# B&R Automation Studio project Y4_V3_1 (part 3)

#### IecCheck.st - Implementation file
```iecst
(********************************************************************
 * COPYRIGHT --
 ********************************************************************
 * Library: IecCheck
 * Author: NickE
 * Created: July 12, 2011
 ********************************************************************
 * Implementation of library IecCheck
 ********************************************************************)

(* Check divisor for DINT and UDINT division *)
FUNCTION CheckDivDWord
	IF divisor=0 THEN
		CheckDivDWord:=1;
	ELSE
		CheckDivDWord:=divisor;
	END_IF
END_FUNCTION

(* Check divisor for INT and UINT division *)
FUNCTION CheckDivWord
	IF divisor=0 THEN
		CheckDivWord:=1;
	ELSE
		CheckDivWord:=divisor;
	END_IF
END_FUNCTION

(* Check divisor for SINT and USINT division *)
FUNCTION CheckDivByte
	IF divisor=0 THEN
		CheckDivByte:=1;
	ELSE
		CheckDivByte:=divisor;
	END_IF
END_FUNCTION

(* Check divisor for REAL division *)
FUNCTION CheckDivReal
	IF divisor=0 THEN
		CheckDivReal:=1;
	ELSE
		CheckDivReal:=divisor;
	END_IF
END_FUNCTION

(* Check divisor for LREAL division *)
FUNCTION CheckDivLReal
	IF divisor=0 THEN
		CheckDivLReal:=1;
	ELSE
		CheckDivLReal:=divisor;
	END_IF
END_FUNCTION

(* Check range for array access *)
FUNCTION CheckBounds
	IF index < lower THEN
		CheckBounds := lower;
	ELSIF index > upper THEN
		CheckBounds := upper;
	ELSE
		CheckBounds := index;
	END_IF
END_FUNCTION

(* Check range for enumeration *)
FUNCTION CheckRange
	IF value < lower THEN
		CheckRange := lower;
	ELSIF value > upper THEN
		CheckRange := upper;
	ELSE
		CheckRange := value;
	END_IF
END_FUNCTION

(* Check address when reading dynamic variables *)
FUNCTION CheckReadAccess
	IF address=0 THEN
		(* TODO: Insert an appropriate code, see AutomationStudio help for further information *)
	END_IF

	CheckReadAccess:=0;
END_FUNCTION

(* Check address when writing dynamic variables *)
FUNCTION CheckWriteAccess
	IF address=0 THEN
		(* TODO: Insert an appropriate code, see AutomationStudio help for further information *)
	END_IF

	CheckWriteAccess:=0;
END_FUNCTION
```

### Library Logical/Libraries/Lib_Ashton (IEC)

#### Lib_Ashton.fun - Exported functions and function blocks
```iecst
(********************************************************************
 * COPYRIGHT --
 ********************************************************************
 * Library: Ashton
 * File: Ashton.fun
 * Author: nicke
 * Created: May 27, 2008
 ********************************************************************
 * Functions and function blocks of library Ashton
 ********************************************************************)

FUNCTION_BLOCK TrackCount (*Count Tracked pieces*)
	VAR_INPUT
		IN1 : USINT; (*Add your parameter comment*)
		IN2 : USINT; (*Add your parameter comment*)
		IN3 : USINT; (*Add your parameter comment*)
		IN4 : USINT; (*Add your parameter comment*)
		IN5 : USINT; (*Add your parameter comment*)
		IN6 : USINT; (*Add your parameter comment*)
	END_VAR
	VAR_OUTPUT
		Count : USINT; (*Add your parameter comment*)
	END_VAR
END_FUNCTION_BLOCK

FUNCTION_BLOCK Photo (*Anti bounce input filter*)
	VAR_INPUT
		SensorIN : BOOL; (*Add your parameter comment*)
		SpeedON : REAL; (*Add your parameter comment*)
		SpeedOFF : REAL; (*Add your parameter comment*)
		OverrideON : UDINT;
		OverrideOFF : UDINT;
	END_VAR
	VAR_OUTPUT
		SensorOUT : BOOL; (*Add your parameter comment*)
		PTON : TIME;
		PTOFF : TIME;
		Measured : REAL;
	END_VAR
	VAR
		Measure : CycleTime_typ;
		DelayB4ON : TON; (*Add your parameter comment*)
		DelayB4OFF : TON; (*Add your parameter comment*)
		zzEdge00000 : BOOL;
		zzEdge00001 : BOOL;
		zzEdge00002 : BOOL;
		zzEdge00003 : BOOL;
	END_VAR
END_FUNCTION_BLOCK

FUNCTION_BLOCK TrackProc (*TODO: Add your comment here*)
	VAR_INPUT
		ONStart : BOOL; (*Add your parameter comment*)
		OFFStart : BOOL; (*Add your parameter comment*)
		EStop : BOOL; (*Add your parameter comment*)
		PT_On : UDINT; (*Add your parameter comment*)
		PT_Off : UDINT; (*Add your parameter comment*)
		End : BOOL;
	END_VAR
	VAR_OUTPUT
		Out : BOOL; (*Add your parameter comment*)
	END_VAR
	VAR
		ON : TON; (*Add your parameter comment*)
		OFF : TON; (*Add your parameter comment*)
		BeforeOn : BOOL;
		BeforeOff : BOOL;
		zzEdge00000 : BOOL;
		zzEdge00001 : BOOL;
		zzEdge00002 : BOOL;
		zzEdge00003 : BOOL;
		zzEdge00004 : BOOL;
		PTOnEStop : TIME;
		PTOffEStop : TIME;
		Recover : BOOL;
		ONPT : TIME;
		OFFPT : TIME;
	END_VAR
END_FUNCTION_BLOCK

FUNCTION_BLOCK C5Restart (*Calculate Restart delay for C5R*)
	VAR_INPUT
		Start : BOOL; (*Add your parameter comment*)
		Speed : REAL; (*Add your parameter comment*)
	END_VAR
	VAR_OUTPUT
		Out : BOOL; (*Add your parameter comment*)
	END_VAR
	VAR
		TON_001 : TON; (*Add your parameter comment*)
		Preset : REAL; (*Add your parameter comment*)
	END_VAR
END_FUNCTION_BLOCK

FUNCTION_BLOCK RunTime (*Calculate system run time*)
	VAR_INPUT
		On : BOOL; (*Add your parameter comment*)
		TotReset : BOOL; (*Total Reset*)
		ShftReset : BOOL; (*Shift Reset*)
		TotMinIn : UINT; (*Total minutes In*)
		TotHrIn : UINT; (*Total hours In*)
		TotDayIn : UINT; (*Total days In*)
		TotYrIn : UINT; (*Total years In*)
		ShftMinIn : UINT; (*Shft minutes In*)
		ShftHrIn : UINT; (*Shift hours In*)
		ShftDayIn : UINT; (*Shift days In*)
		ShftYrIn : UINT; (*Shift years In*)
	END_VAR
	VAR_OUTPUT
		TotMin : UINT; (*Total Minutes*)
		TotHr : UINT; (*Total Hours*)
		TotDay : UINT; (*Total Days*)
		TotYr : UINT; (*Total Years*)
		ShftMin : UINT; (*Shift Minutes*)
		ShftHr : UINT; (*Shift Hours*)
		ShftDay : UINT; (*Shift Days*)
		ShftYr : UINT; (*Shift Years*)
	END_VAR
	VAR
		Minute : TON; (*Minute timer*)
	END_VAR
END_FUNCTION_BLOCK

FUNCTION_BLOCK GrindTime (*Calculate grind time and length*)
	VAR_INPUT
		On : BOOL; (*Start trigger*)
		TotReset : BOOL; (*Total Reset*)
		ShftReset : BOOL; (*Shift Reset*)
		Speed : REAL; (*Seaming speed*)
		Measured : REAL; (*Measured length/width*)
		TotMSIn : UINT; (*Total Milliseconds*)
		TotSecIn : UINT; (*Total Seconds*)
		TotMinIn : UINT; (*Total Minutes*)
		TotHrIn : UINT; (*Total Hours*)
		TotDayIn : UINT; (*Total Days*)
		ShftMSIn : UINT; (*Shift Milliseconds*)
		ShftSecIn : UINT; (*Shift Seconds*)
		ShftMinIn : UINT; (*Shift Minutes*)
		ShftHrIn : UINT; (*Shift Hours*)
		ShftDayIn : UINT; (*Shift Days*)
		TotMtrs1In : UDINT; (*Total Meters 1*)
		TotMtrs2In : UDINT; (*Total Meters 2*)
		TotFt1In : UDINT; (*Total Feet 1*)
		TotFt2In : UDINT; (*Total Feet 2*)
		ShftMtrs1In : UDINT; (*Shift Meters 1*)
		ShftMtrs2In : UDINT; (*Shift Meters 2*)
		ShftFt1In : UDINT; (*Shift Feet 1*)
		ShftFt2In : UDINT; (*Shift Feet 2*)
	END_VAR
	VAR_OUTPUT
		TotMS : UINT; (*Total Milliseconds*)
		TotSec : UINT; (*Total Seconds*)
		TotMin : UINT; (*Total Minutes*)
		TotHr : UINT; (*Total Hours*)
		TotDay : UINT; (*Total Days*)
		ShftMS : UINT; (*Shift Milliseconds*)
		ShftSec : UINT; (*Shift Seconds*)
		ShftMin : UINT; (*Shift Minutes*)
		ShftHr : UINT; (*Shift Hours*)
		ShftDay : UINT; (*Shift Days*)
		TotMtrs1 : UDINT; (*Total Meters 1*)
		TotMtrs2 : UDINT; (*Total Meters 2*)
		TotFt1 : UDINT; (*Total Feet 1*)
		TotFt2 : UDINT; (*Total Feet 2*)
		ShftMtrs1 : UDINT; (*Shift Meters 1*)
		ShftMtrs2 : UDINT; (*Shift Meters 2*)
		ShftFt1 : UDINT; (*Shift Feet 1*)
		ShftFt2 : UDINT; (*Shift Feet 2*)
	END_VAR
	VAR
		CurrentMS : REAL; (*Current measured length in millisec*)
		WholeSec : UINT; (*Calculated whole seconds*)
		CurrentMSUINT : UINT; (*CurrentMS in UINT*)
		WholeMSec : UINT;
		Calc3 : UINT;
		MeasuredFtUD : UDINT; (*Measured feet UDINT*)
		MeasuredUD : UDINT; (*Measured Mtrs UDINT*)
		MeasuredM : REAL; (*Measured Mtrs*)
		MeasuredFt : REAL; (*Measured feet*)
		zzEdge00000 : BOOL;
	END_VAR
END_FUNCTION_BLOCK

FUNCTION_BLOCK Center2 (*TODO: Add your comment here*)
	VAR_INPUT
		WidthIn : REAL; (*Add your parameter comment*)
		Speed : REAL; (*Add your parameter comment*)
		Centre : REAL; (*Add your parameter comment*)
	END_VAR
	VAR_OUTPUT
		PT : UDINT; (*Add your parameter comment*)
	END_VAR
	VAR
		Calc1 : REAL; (*Add your parameter comment*)
		DecTime : REAL; (*Add your parameter comment*)
		DecDist : REAL; (*Add your parameter comment*)
		PTReal : REAL; (*Add your parameter comment*)
	END_VAR
END_FUNCTION_BLOCK

FUNCTION_BLOCK Center (*TODO: Add your comment here*)
	VAR_INPUT
		WidthIn : REAL; (*Add your parameter comment*)
		Speed : REAL; (*Add your parameter comment*)
		Centre : REAL; (*Add your parameter comment*)
	END_VAR
	VAR_OUTPUT
		PT : UDINT; (*Add your parameter comment*)
	END_VAR
	VAR
		Calc1 : REAL; (*Add your parameter comment*)
		AccTime : REAL; (*Add your parameter comment*)
		AccDecDist : REAL; (*Add your parameter comment*)
		PTReal : REAL; (*Add your parameter comment*)
	END_VAR
END_FUNCTION_BLOCK

FUNCTION_BLOCK TrackBit (*Tracking Bit Controls*) (*$GROUP=User,$CAT=User,$GROUPICON=User.png,$CATICON=User.png*)
	VAR_INPUT
		FixedIN : TrackBit_Fixed_typ;
		RunBlock : BOOL;
		SolBlock : BOOL;
		Analog : FB_ANALOG_enum;
		Speed : REAL;
		SpeedAnalog : REAL;
		SpeedMatchEN : BOOL;
		SpeedMatch : REAL;
		TimeoutBlock : BOOL;
		TimeoutEN : BOOL;
		TrackDelayEN : BOOL;
		DelayPT : UDINT;
		TimeoutACK : BOOL;
		DoneIN : BOOL;
	END_VAR
	VAR_OUTPUT
		Active : BOOL;
		Done : BOOL;
		Disp : Display_enum;
		ESDisp : {REDUND_UNREPLICABLE} Display_enum;
		RunOUT : BOOL;
		SolOUT : BOOL;
		SpeedOUT : REAL;
		TimeoutOUT : BOOL;
	END_VAR
	VAR
		DelayTON : TON;
		TimeoutACKLatch : BOOL;
	END_VAR
END_FUNCTION_BLOCK

FUNCTION_BLOCK TrackingSection (*TRACKING SECTION CONTROLS*) (*$GROUP=User,$CAT=User,$GROUPICON=User.png,$CATICON=User.png*)
	VAR_INPUT
		ControlIN : BOOL;
		ESClear : BOOL;
		Cleared : BOOL;
		EMOStart : BOOL;
		Blocks : ARRAY[0..12] OF BOOL;
		BlockInhib : BOOL;
		ResES : BOOL;
		ResMan : BOOL;
		ESDispInhib : BOOL;
		IndexIN : USINT;
		WidthIN : REAL;
		LengthIN : REAL;
		BatchClearIN : BOOL;
		LongestIN : REAL;
		RowBlockIN : BOOL;
		ChangeIN : BOOL;
		ArrissUpperIN : BOOL;
		ArrissLowerIN : BOOL;
		EdgeDeleteIN : BOOL;
		VerticalBeltIN : BOOL;
	END_VAR
	VAR_OUTPUT
		FixedOUT : TrackBit_Fixed_typ;
		Blocked : BOOL;
		Busy : BOOL;
		Index : USINT;
		Width : REAL;
		Length : REAL;
		BatchClear : BOOL;
		Longest : REAL;
		RowBlock : BOOL;
		Change : BOOL;
		ArrissUpper : BOOL;
		ArrissLower : BOOL;
		EdgeDelete : BOOL;
		VerticalBelt : BOOL;
		Cycle : REAL;
		BusyDisp : Display_enum;
	END_VAR
	VAR
		CurrentTime : TIME;
		PreviousTime : TIME;
		ElapsedTime : UDINT;
		i : INT;
		zzEdge00000 : BOOL;
	END_VAR
END_FUNCTION_BLOCK

FUNCTION_BLOCK ControlFB
	VAR_INPUT
		Start : BOOL;
		Stop : BOOL;
		EStop1 : BOOL;
		EStop2 : BOOL;
		BuzzBlock : BOOL;
		StandbyBlock : BOOL;
		Auto : BOOL;
		Test : BOOL;
		ESClear : BOOL;
		Paused : BOOL;
		Alarm : BOOL;
		Warning : BOOL;
		CountIN : ARRAY[0..19] OF BOOL;
		BuzzerPT : UDINT;
		StandbyPT : UDINT;
	END_VAR
	VAR_OUTPUT
		Achieved1 : BOOL;
		Achieved2 : BOOL;
		Buzzer : BOOL;
		Empty : BOOL;
		OnLmp1 : BOOL;
		OnLmp2 : BOOL;
		GrnLmp : BOOL;
		YelLmp : BOOL;
		RedLmp : BOOL;
	END_VAR
	VAR
		BuzzerTON : TON;
		StandbyTON : TON;
		Grn : ARRAY[0..2] OF BOOL;
		Yel : ARRAY[0..2] OF BOOL;
		Red : ARRAY[0..2] OF BOOL;
		TSecOff : BOOL;
		TSecOn : BOOL;
		TSecOFF : TON;
		TSecON : TON;
		StopLatch : BOOL;
		StopDone : BOOL;
		i : USINT;
		zzEdge1 : BOOL;
		zzEdge2 : BOOL;
		zzEdge3 : BOOL;
		zzEdge4 : BOOL;
		zzEdge5 : BOOL;
		EStopStartTON : TON;
		zzEdge6 : BOOL;
		zzEdge7 : BOOL;
		zzEdge00000 : BOOL;
		zzEdge00001 : BOOL;
		zzEdge00002 : BOOL;
		zzEdge00003 : BOOL;
		zzEdge00004 : BOOL;
		zzEdge00005 : BOOL;
		zzEdge00006 : BOOL;
	END_VAR
END_FUNCTION_BLOCK

FUNCTION_BLOCK SeamersFB
	VAR_INPUT
		Enable : ARRAY[0..4] OF BOOL;
		AutoStart : ARRAY[0..4] OF BOOL;
		ESClear : BOOL;
		ControlIN : BOOL;
		EDOn : BOOL;
		TransportMode : BOOL;
		Detension : BOOL;
		Trips : ARRAY[0..24] OF BOOL;
		Float : ARRAY[0..2] OF BOOL;
		BeltsPT : UDINT;
		VacPT : UDINT;
		EDPT : UDINT;
		ExtractionPT : UDINT;
		PumpPT : ARRAY[0..4] OF UDINT;
		VacsStopPT : UDINT;
	END_VAR
	VAR_OUTPUT
		StartAllDisp : Display_enum;
		BeltOUT : ARRAY[0..12] OF BOOL;
		VacOUT : ARRAY[0..4] OF BOOL;
		EDOUT : ARRAY[0..4] OF BOOL;
		ExtractionOUT : ARRAY[0..4] OF BOOL;
		PumpOUT : ARRAY[0..2] OF BOOL;
		DoneOUT : ARRAY[0..4] OF BOOL;
	END_VAR
	VAR
		zzEdge00000 : BOOL;
		zzEdge00001 : BOOL;
		zzEdge00002 : BOOL;
		zzEdge00003 : BOOL;
		zzEdge00004 : BOOL;
		zzEdge00005 : BOOL;
		zzEdge00006 : BOOL;
		zzEdge00007 : BOOL;
		zzEdge00008 : BOOL;
		zzEdge00009 : BOOL;
		zzEdge00010 : BOOL;
		zzEdge00011 : BOOL;
		zzEdge00012 : BOOL;
		zzEdge00013 : BOOL;
		zzEdge00014 : BOOL;
		zzEdge00015 : BOOL;
		zzEdge00016 : BOOL;
		zzEdge00017 : BOOL;
		zzEdge00018 : BOOL;
		zzEdge00019 : BOOL;
		zzEdge00020 : BOOL;
		zzEdge00021 : BOOL;
		zzEdge00022 : BOOL;
		zzEdge00023 : BOOL;
		zzEdge00024 : BOOL;
		zzEdge00025 : BOOL;
		zzEdge00026 : BOOL;
		zzEdge00027 : BOOL;
		Latch : BOOL;
		LatchES : BOOL;
		Starting1 : BOOL;
		Starting2 : BOOL;
		Starting3 : BOOL;
		Starting4 : BOOL;
		Belt1TON : TON;
		Belt2TON : TON;
		Belt3TON : TON;
		Belt4TON : TON;
		Belt5TON : TON;
		Belt6TON : TON;
		Belt7TON : TON;
		Belt8TON : TON;
		Belt9TON : TON;
		Belt10TON : TON;
		Belt11TON : TON;
		Belt12TON : TON;
		ED1TON : TON;
		ED2TON : TON;
		ED3TON : TON;
		ED4TON : TON;
		Vac1TON : TON;
		Vac2TON : TON;
		Vac3TON : TON;
		Vac4TON : TON;
		Extract1TON : TON;
		Extract2TON : TON;
		Extract3TON : TON;
		Extract4TON : TON;
		Pump4TON : TON;
		Pump3TON : TON;
		Pump1TON : TON;
		Pump2TON : TON;
		i : INT;
		VacStopTON : TON;
		zzEdge00028 : BOOL;
		zzEdge00029 : BOOL;
		zzEdge00030 : BOOL;
		zzEdge00031 : BOOL;
	END_VAR
END_FUNCTION_BLOCK

FUNCTION_BLOCK InvTestFB
	VAR_INPUT
		Index : USINT;
		AutoSpeedIN : REAL;
		SpeedIN : PLInvPerm;
		TestSpeedIN : REAL;
		AnalogSpeedIN : REAL;
	END_VAR
	VAR_OUTPUT
		Run : BOOL;
		Rev : BOOL;
		Speed : REAL;
	END_VAR
END_FUNCTION_BLOCK

FUNCTION_BLOCK Batch (*ROW BUILDING CALCULATIONS*) (*$GROUP=User,$CAT=User,$GROUPICON=User.png,$CATICON=User.png*)
	VAR_INPUT
		Calculate : BOOL;
		ClearIN : BOOL;
		Building : BOOL;
		Gap : REAL;
		MaxSize : REAL;
		CenterDist : REAL;
		CenterSpeed : REAL;
		FollowingIN : ARRAY[0..9] OF REAL;
		LengthIN : REAL;
		BatchMode : BATCHING_enum;
		Type : BATCHTYPE_enum;
	END_VAR
	VAR_OUTPUT
		Longest : REAL;
		Current : REAL;
		Next : REAL;
		Done : BOOL;
		CenterPT : UDINT;
		Remaining : REAL;
	END_VAR
	VAR
		i : USINT;
		MinRemaining : REAL;
		NextSize : REAL;
		NextLengthINT : REAL;
		NextINT : REAL;
		DoubleCount : USINT;
		Center : Center;
		zzEdge00000 : BOOL;
		zzEdge00001 : BOOL;
		zzEdge00002 : BOOL;
		zzEdge00003 : BOOL;
		zzEdge00004 : BOOL;
		zzEdge00005 : BOOL;
		zzEdge00006 : BOOL;
		zzEdge00007 : BOOL;
		zzEdge00008 : BOOL;
		zzEdge00009 : BOOL;
	END_VAR
END_FUNCTION_BLOCK

FUNCTION_BLOCK SeamersSMProFB (*Seamers start up control SMPro*) (*$GROUP=User,$CAT=User,$GROUPICON=User.png,$CATICON=User.png*)
	VAR_INPUT
		Enable : ARRAY[0..4] OF BOOL;
		AutoStart : ARRAY[0..4] OF BOOL;
		ESClear : BOOL;
		ControlIN : BOOL;
		EDOn : BOOL;
		TransportMode : BOOL;
		Detension : BOOL;
		Trips : ARRAY[0..24] OF BOOL;
		Float : ARRAY[0..2] OF BOOL;
		BeltsPT : UDINT;
		VacPT : UDINT;
		EDPT : UDINT;
		ExtractionPT : UDINT;
		PumpPT : ARRAY[0..4] OF UDINT;
		VacsStopPT : UDINT;
	END_VAR
	VAR_OUTPUT
		StartAllDisp : Display_enum;
		BeltOUT : ARRAY[0..12] OF BOOL;
		VacOUT : ARRAY[0..4] OF BOOL;
		EDOUT : ARRAY[0..4] OF BOOL;
		ExtractionOUT : ARRAY[0..4] OF BOOL;
		PumpOUT : ARRAY[0..2] OF BOOL;
		DoneOUT : ARRAY[0..4] OF BOOL;
	END_VAR
	VAR
		Latch : BOOL;
		LatchES : BOOL;
		Starting1 : BOOL;
		Starting2 : BOOL;
		Belt1TON : TON;
		Belt2TON : TON;
		Belt3TON : TON;
		Belt4TON : TON;
		Belt5TON : TON;
		Belt6TON : TON;
		Belt7TON : TON;
		Belt8TON : TON;
		Belt9TON : TON;
		Belt10TON : TON;
		Belt11TON : TON;
		Belt12TON : TON;
		ED1TON : TON;
		ED2TON : TON;
		ED3TON : TON;
		ED4TON : TON;
		Vac1TON : TON;
		Vac2TON : TON;
		Vac3TON : TON;
		Vac4TON : TON;
		Extract1TON : TON;
		Extract2TON : TON;
		Extract3TON : TON;
		Extract4TON : TON;
		Pump4TON : TON;
		Pump3TON : TON;
		Pump1TON : TON;
		Pump2TON : TON;
		i : INT;
		VacStopTON : TON;
		zzEdge00000 : BOOL;
		zzEdge00001 : BOOL;
		zzEdge00002 : BOOL;
		zzEdge00003 : BOOL;
		zzEdge00004 : BOOL;
		zzEdge00005 : BOOL;
		zzEdge00006 : BOOL;
		zzEdge00007 : BOOL;
		zzEdge00008 : BOOL;
		zzEdge00009 : BOOL;
		zzEdge00010 : BOOL;
		zzEdge00011 : BOOL;
		zzEdge00012 : BOOL;
		zzEdge00013 : BOOL;
		zzEdge00014 : BOOL;
		zzEdge00015 : BOOL;
		zzEdge00016 : BOOL;
		zzEdge00017 : BOOL;
	END_VAR
END_FUNCTION_BLOCK

FUNCTION_BLOCK FlipUps (*FLIP UP ARMS CONTROL*) (*$GROUP=User,$CAT=User,$GROUPICON=User.png,$CATICON=User.png*)
	VAR_INPUT
		ActPos : REAL; (*Seamer Actual Position*)
		ArmPos : ARRAY[0..5] OF REAL; (*Arm Actual Positions*)
		Up : ARRAY[0..10] OF BOOL; (*Array for arms up reed switches*)
		i : INT; (*Index for FOR loops*)
		Down : ARRAY[0..10] OF BOOL; (*Array for arms down reed switches*)
		HiVol : BOOL; (*Mode Selection*)
		Arms : USINT; (*Number of Arms*)
		Raise : BOOL; (*Condition to raise arms*)
	END_VAR
	VAR_OUTPUT
		UpDone : BOOL; (*Selected arms up*)
		OUT : ARRAY[0..5] OF BOOL; (*Raise Arms Output*)
		DownDone : BOOL; (*All arms down*)
		CheckRaised : INT; (*Number of arms to raise*)
	END_VAR
	VAR
		zzEdge00000 : BOOL;
	END_VAR
END_FUNCTION_BLOCK

FUNCTION_BLOCK NozzleControl (*TODO: Add your comment here*) (*$GROUP=User,$CAT=User,$GROUPICON=User.png,$CATICON=User.png*)
	VAR_INPUT
		PreTrack : ARRAY[0..2] OF BOOL; (*[0] = Blocked [1..2] Pre track bits, during S&F and ready and block conditions off*)
		Track : ARRAY[0..6] OF BOOL; (*TrackBits when nozzles to be active*)
		VacuumStopDelay : UDINT; (*Vacuum Stop delay after Control Stop*)
		NozzlePerm : NozzlePerm_typ; (*NozzlePerm.OpenDelay/PurgeCount*)
		Vacuum : BOOL; (*Link to 2nd pump running before nozzles on*)
		AutoStart : BOOL; (*Seamer specific AutoStart condition*)
		Control : BOOL; (*Control.Achieved1*)
		TransportMode : BOOL; (*Seamers.TransportMode*)
		PreTracking : INT; (*Pretracking number, used to turn on spray earlier if required*)
	END_VAR
	VAR_OUTPUT
		Spray : BOOL; (*Spray solenoid output control*)
		ControlStop : INT; (*ControlStop count for current power cycle*)
		Nozzle : NozzleControl_typ; (*Start up and stop sequence control*)
	END_VAR
	VAR
		IdleIntervalTON : TON; (*If track off for period*)
		IdleOpenTON : TON; (*Open delay if idle*)
		TrackIndex : USINT; (*For loop index of Track*)
		SequenceIO : IntervalOpen_enum;
	END_VAR
END_FUNCTION_BLOCK

FUNCTION_BLOCK SeamersSMProIIFB (*TODO: Add your comment here*) (*$GROUP=User,$CAT=User,$GROUPICON=User.png,$CATICON=User.png*)
	VAR_INPUT
		Enable : ARRAY[0..2] OF BOOL;
		AutoStart : ARRAY[0..2] OF BOOL;
		EDOn : BOOL;
		TransportMode : BOOL;
		Detension : BOOL;
		Trips : ARRAY[0..80] OF BOOL;
		SeekBlock : ARRAY[0..2] OF BOOL;
		Float : ARRAY[0..2] OF BOOL;
		Shaker : BOOL;
		PresetSys : Preset_Seamers_typ;
		InterceptOpen : UDINT;
		InterceptInterval : UDINT;
		Control : Control_typ;
	END_VAR
	VAR_OUTPUT
		StartAllDisp : Display_enum;
		BeltOUT : ARRAY[0..12] OF BOOL;
		VacOUT : ARRAY[0..4] OF BOOL;
		EDOUT : ARRAY[0..4] OF BOOL;
		ExtractionOUT : ARRAY[0..4] OF BOOL;
		PumpOUT : ARRAY[0..2] OF BOOL;
		ValveOUT : ARRAY[0..2] OF BOOL;
		DoneOUT : ARRAY[0..4] OF BOOL;
		BackGround : Control_BackGround_typ;
	END_VAR
	VAR
		AutoStart1 : SeamerStart_enum;
		AutoStart2 : SeamerStart_enum;
		Latch : BOOL;
		LatchES : BOOL;
		Starting1 : BOOL;
		Starting2 : BOOL;
		Scavenge : Interval_typ;
		Belt1TON : TON;
		Belt2TON : TON;
		Belt3TON : TON;
		Belt4TON : TON;
		Belt5TON : TON;
		Belt6TON : TON;
		Belt7TON : TON;
		Belt8TON : TON;
		Belt9TON : TON;
		Belt10TON : TON;
		Belt11TON : TON;
		Belt12TON : TON;
		ED1TON : TON;
		ED2TON : TON;
		ED3TON : TON;
		ED4TON : TON;
		Vac1TON : TON;
		Vac2TON : TON;
		Vac3TON : TON;
		Vac4TON : TON;
		Extract1TON : TON;
		Extract2TON : TON;
		Extract3TON : TON;
		Extract4TON : TON;
		Pump4TON : TON;
		Pump3TON : TON;
		Pump1TON : TON;
		Pump2TON : TON;
		i : INT;
		VacuumRunOn : VacuumRunOn_enum;
		InterceptOpen2TON : TON;
		InterceptOpen1TON : TON;
		InterceptInterval2TON : TON;
		InterceptInterval1TON : TON;
		Intercept2 : IntervalDelay_enum;
		Intercept1 : IntervalDelay_enum;
		VacStopTON : TON;
		zzEdge00000 : BOOL;
	END_VAR
END_FUNCTION_BLOCK
```

#### TrackCount.st
```iecst
(********************************************************************
 * COPYRIGHT --
 ********************************************************************
 * Library: Ashton
 * File: TrackCount.st
 * Author: nicke
 * Created: May 27, 2008
 ********************************************************************
 * Implementation of library Ashton
 ********************************************************************)

(*TODO: Add your comment here*)
FUNCTION_BLOCK TrackCount

	Count:= 0;

	IF IN1 > 0 THEN
		Count:= Count + 1;
	END_IF
	IF IN2 > 0 THEN
		Count:= Count + 1;
	END_IF
	IF IN3 > 0 THEN
		Count:= Count + 1;
	END_IF
	IF IN4 > 0 THEN
		Count:= Count + 1;
	END_IF
	IF IN5 > 0 THEN
		Count:= Count + 1;
	END_IF
	IF IN6 > 0 THEN
		Count:= Count + 1;
	END_IF

END_FUNCTION_BLOCK
```

#### Photo.st - Anti bounce input filter
```iecst
(********************************************************************
 * COPYRIGHT --
 ********************************************************************
 * Library: Ashton
 * File: Photo.st
 * Author: nicke
 ********************************************************************
 * Implementation of library Ashton
 ********************************************************************)

//ANTI BOUNCE INPUT FILTER
FUNCTION_BLOCK Photo

	//TON DelayB4ON USED TO TURN ON INTERNAL INPUT
	//FB INPUTS
	DelayB4ON.IN := SensorIN ;
	PTON := UDINT_TO_TIME(REAL_TO_UDINT(1200/SpeedON)) ;
	IF(OverrideON = 0) THEN
		DelayB4ON.PT := PTON ;
	ELSE
		DelayB4ON.PT := OverrideON ;
	END_IF
	//CALL FB
	DelayB4ON ();
	//FB OUTPUT
	IF EDGEPOS(DelayB4ON.Q) THEN
		SensorOUT := TRUE;
	END_IF

	//TON DelayB4OFF USED TO TURN OFF INTERNAL INPUT
	//FB INPUTS
	DelayB4OFF.IN := NOT(SensorIN) ;
	PTOFF := UDINT_TO_TIME(REAL_TO_UDINT(1200/SpeedOFF)) ;
	IF(OverrideOFF = 0) THEN
		DelayB4OFF.PT := PTOFF ;
	ELSE
		DelayB4OFF.PT := OverrideOFF ;
	END_IF
	//CALL FB
	DelayB4OFF ();
	//FB OUTPUT
	IF EDGEPOS(DelayB4OFF.Q) THEN
		SensorOUT := FALSE;
	END_IF

	//SENSOR ELAPSED TIME - USED FOR MEASUREMENT CALCULATION
	IF EDGEPOS(SensorOUT) THEN
		Measure.Previous := clock_ms() ;
	END_IF
	IF EDGENEG(SensorOUT) THEN
		Measure.Current := clock_ms() ;
		Measure.Elapsed := TIME_TO_UDINT(Measure.Current - Measure.Previous) ;
	END_IF
	Measured := (UDINT_TO_REAL(Measure.Elapsed))*(SpeedON/60) ;

END_FUNCTION_BLOCK
```

#### TrackProc.st
```iecst
(********************************************************************
 * COPYRIGHT --
 ********************************************************************
 * Library: Ashton
 * File: TrackProc.st
 * Author: nicke
 * Created: June 03, 2008
 ********************************************************************
 * Implementation of library Ashton
 ********************************************************************)

(*Process Tracking Register*)
FUNCTION_BLOCK TrackProc

(*At EStop capture elapsed time and creat new preset time*)
IF EDGEPOS(EStop) THEN
	PTOnEStop:= (UDINT_TO_TIME(PT_On) - ON.ET);
	PTOffEStop:= (UDINT_TO_TIME(PT_Off) - OFF.ET);
	Recover:= TRUE;
END_IF

IF NOT(Recover) THEN
	ONPT:= UDINT_TO_TIME(PT_On);
	OFFPT:= UDINT_TO_TIME(PT_Off);
ELSE
	ONPT:= PTOnEStop;
	OFFPT:= PTOffEStop;
END_IF

(* Check for On Start Condition*)
IF EDGEPOS(ONStart) THEN
	BeforeOn:= TRUE;
END_IF

(* Time delay before process on*)
ON( IN:= (BeforeOn AND NOT EStop), PT:= ONPT);

IF EDGEPOS(ON.Q) THEN
	Out:= TRUE;
	BeforeOn:= FALSE;
END_IF

(* Check for Off Start Condition*)
IF EDGEPOS(OFFStart) THEN
	BeforeOff:= TRUE;
END_IF

(* Time delay before process off*)
OFF( IN:= (BeforeOff AND NOT EStop), PT:= OFFPT);

IF EDGEPOS(OFF.Q) THEN
	Out:= FALSE;
	BeforeOff:= FALSE;
END_IF

IF (End) THEN
	BeforeOn:= FALSE;
	BeforeOff:= FALSE;
	Recover:= FALSE;
	Out:= FALSE;
END_IF

END_FUNCTION_BLOCK
```

#### C5Restart.st - Calculate Restart delay for C5R
```iecst
(********************************************************************
 * COPYRIGHT --
 ********************************************************************
 * Library: Ashton
 * File: C5Restart.st
 * Author: nicke
 * Created: June 05, 2008
 ********************************************************************
 * Implementation of library Ashton
 ********************************************************************)

(*Calculate Restart delay for C5R*)
FUNCTION_BLOCK C5Restart
(* Calculate valus for preset *)
Preset:= (6000/(Speed/6));
IF Preset < 3000.0 THEN
	Preset:= 1.0;
ELSE
	Preset:= (Preset - 3000.0);
END_IF

(* Delay for C5 restart *)
TON_001( IN:= Start, PT:= UDINT_TO_TIME(REAL_TO_UDINT(Preset)) );
Out:= TON_001.Q;

END_FUNCTION_BLOCK
```

#### RunTime.st - Calculate system run time
```iecst
(********************************************************************
 * COPYRIGHT --
 ********************************************************************
 * Library: Ashton
 * File: RunTime.st
 * Author: NickE
 * Created: June 09, 2008
 ********************************************************************
 * Implementation of library Ashton
 ********************************************************************)

(*Calculate system run time*)
FUNCTION_BLOCK RunTime

(* Write retained values to Internal UINT data *)
TotMin:= TotMinIn;
TotHr:= TotHrIn;
TotDay:= TotDayIn;
TotYr:= TotYrIn;
ShftMin:= ShftMinIn;
ShftHr:= ShftHrIn;
ShftDay:= ShftDayIn;
ShftYr:= ShftYrIn;

(*Count Run Time minutes*)
Minute( IN:= On AND NOT Minute.Q, PT:= T#1m);
IF (Minute.Q) THEN
	TotMin := TotMin+1;
	ShftMin:= ShftMin+1;
END_IF

(*Calculate Total Run Time Hours*)
IF TotMin = 60 THEN
	TotHr := TotHr+1;
	TotMin := 0;
END_IF
(*Calculate Shift Run Time Hours*)
IF ShftMin = 60 THEN
	ShftHr := ShftHr +1;
	ShftMin := 0;
END_IF
(*Calculate Total Run Time Days*)
IF TotHr = 24 THEN
	TotDay := TotDay + 1;
	TotHr := 0;
END_IF
(*Calculate Shift Run Time Days*)
IF ShftHr = 24 THEN
	ShftDay := ShftDay + 1;
	ShftHr := 0;
END_IF
(*Calculate Total Run Time Years*)
IF TotDay = 365 THEN
	TotYr := TotYr + 1;
	TotDay := 0;
END_IF;
(*Calculate Shift Run Time Years*)
IF ShftDay = 365 THEN
	ShftYr := ShftYr +1;
	ShftDay := 0;
END_IF;
(*Reset Shift Values*)
IF (ShftReset) THEN
	ShftMin:= 0;
	ShftHr:= 0;
	ShftDay:=0;
	ShftYr:=0;
END_IF;
(*Reset Total Values*)
IF TotReset = TRUE THEN
	TotMin:= 0;
	TotHr:= 0;
	TotDay:=0;
	TotYr:=0;
END_IF;

END_FUNCTION_BLOCK
```

#### GrindTime.st - Calculate grind time and length
```iecst
(********************************************************************
 * COPYRIGHT --
 ********************************************************************
 * Library: Ashton
 * File: GrindTime.st
 * Author: nicke
 * Created: June 09, 2008
 ********************************************************************
 * Implementation of library Ashton
 ********************************************************************)

(*Calculate grind time and length*)
FUNCTION_BLOCK GrindTime

TotMS:= TotMSIn;
TotSec:= TotSecIn;
TotMin:= TotMinIn;
TotHr:= TotHrIn;
TotDay:= TotDayIn;
ShftMS:= ShftMSIn;
ShftSec:= ShftSecIn;
ShftMin:= ShftMinIn;
ShftHr:= ShftHrIn;
ShftDay:= ShftDayIn;
TotMtrs1:= TotMtrs1In;
TotMtrs2:= TotMtrs2In;
TotFt1:= TotFt1In;
TotFt2:= TotFt2In;
ShftMtrs1:= ShftMtrs1In;
ShftMtrs2:= ShftMtrs2In;
ShftFt1:= ShftFt1In;
ShftFt2:= ShftFt2In;

(* Enable calculation only when not resetting*)
IF EDGEPOS(On) AND NOT(TotReset) AND NOT(ShftReset) THEN
	(*Convert Measured Length/Width into msec*)
	CurrentMS:= Measured/(Speed/60.0);
	(*Convert to UINT value to split into whole seconds and milliseconds under 1000*)
	CurrentMSUINT:= REAL_TO_UINT (CurrentMS);
	WholeSec:=CurrentMSUINT/1000;
	Calc3:=WholeSec*1000;
	WholeMSec:=CurrentMSUINT-Calc3;

	(*Add milliseconds to Total Milliseconds*)
	TotMS:=WholeMSec+TotMS;

	IF TotMS>=1000 THEN
		TotMS:=TotMS-1000;
		TotSec:=TotSec+WholeSec+1;
	ELSE
		TotSec:=TotSec+WholeSec;
	END_IF

		(*Add milliseconds to Temporary Milliseconds*)
	ShftMS:=WholeMSec+ShftMS;

	IF ShftMS>=1000 THEN
		ShftMS:=ShftMS-1000;
		ShftSec:=ShftSec+WholeSec+1;
	ELSE
		ShftSec:=ShftSec+WholeSec;
	END_IF

	(*Calculate Machine Grind Time Minutes*)
	IF TotSec >= 60 THEN
		TotMin:=TotMin + 1;
		TotSec:= TotSec-60;
	END_IF
	IF ShftSec >= 60 THEN
		ShftMin:=ShftMin + 1;
		ShftSec:= ShftSec-60;
	END_IF
	(*Calculate Machine Grind Time Hours*)
	IF TotMin >= 60 THEN
		TotHr:=TotHr + 1;
		TotMin:= TotMin-60;
	END_IF
	IF ShftMin >= 60 THEN
		ShftHr:=ShftHr + 1;
		ShftMin:=ShftMin-60;
	END_IF
	(*Calculate Machine Grind Time Days*)
	IF TotHr >= 24 THEN
		TotDay:=TotDay + 1;
		TotHr:= TotHr-24;
	END_IF
	IF ShftHr = 24 THEN
		ShftDay:=ShftDay + 1;
		ShftHr:= ShftHr-24;
	END_IF

	(*Calculate grind length for belt wear calculations*)
	MeasuredM:= Measured;
	MeasuredUD:= REAL_TO_UDINT(MeasuredM);
	TotMtrs1:= MeasuredUD + TotMtrs1;
	IF TotMtrs1>= 1000000000 THEN
		TotMtrs2:= TotMtrs2+1;
		TotMtrs1:= TotMtrs1 - 1000000000;
	END_IF

	ShftMtrs1:= MeasuredUD + ShftMtrs1;
	IF ShftMtrs1>= 1000000000 THEN
		ShftMtrs2:= ShftMtrs2+1;
		ShftMtrs1:= ShftMtrs1 - 1000000000;
	END_IF

	(*Calculate grind length in Feet*)
	MeasuredFt:= MeasuredM * 3048.0;
	MeasuredFtUD:= REAL_TO_UDINT (MeasuredFt);
	TotFt1:= MeasuredFtUD + TotFt1;
	IF TotFt1>= 1000000000 THEN
		TotFt2:= TotFt2+1;
		TotFt1:= TotFt1 - 1000000000;
	END_IF

	ShftFt1:= MeasuredFtUD + ShftFt1;
	IF ShftFt1>= 1000000000 THEN
		ShftFt2:= ShftFt2+1;
		ShftFt1:= ShftFt1 - 1000000000;
	END_IF

END_IF

(*Reset Total Values*)
IF TotReset = TRUE THEN
	TotMS:= 0;
	TotSec:=0;
	TotMin:=0;
	TotHr:=0;
	TotDay:=0;
	TotMtrs1:= 0;
	TotMtrs2:= 0;
	TotFt1:= 0;
	TotFt2:= 0;
END_IF
IF ShftReset = TRUE THEN
	ShftMS:=0;
	ShftSec:=0;
	ShftMin:=0;
	ShftHr:=0;
	ShftDay:=0;
	ShftMtrs1:= 0;
	ShftMtrs2:= 0;
	ShftFt1:= 0;
	ShftFt2:= 0;
END_IF

END_FUNCTION_BLOCK
```

#### Center.st
```iecst
(********************************************************************
 * COPYRIGHT --
 ********************************************************************
 * Library: Ashton
 * File: Center.st
 * Author: nicke
 ********************************************************************
 * Implementation of library Ashton
 ********************************************************************)

//CALCULATE PRESET TIME FOR CENTERING
FUNCTION_BLOCK Center

	//CALCULATE M/MIN
	Calc1 := Speed / 60 ;
	//CALCULATE TIME REQUIRED FOR ACCELERATION
	AccTime := (Calc1 * 0.5) * 100 ;
	//CALCULATE DISTANCE TRAVELLED DURING ACCELERATION AND DECELERATION
	AccDecDist := (((Calc1 / 4) * Calc1) * 2) * 1000 ;
	//CALCULATE PRESET TIME FOR BATCH CENTERING TIME DELAY
	PTReal:=(((Centre - (WidthIn / 2) - AccDecDist) / Calc1) / 10) + AccTime ;
	//CONVERT REAL VALUE INTO UDINT
	PT := REAL_TO_UDINT (PTReal) ;

END_FUNCTION_BLOCK
```

#### Center2.st
```iecst
(********************************************************************
 * COPYRIGHT --
 ********************************************************************
 * Library: Ashton
 * File: Center.st
 * Author: nicke
 * Created: September 09, 2009
 ********************************************************************
 * Implementation of library Ashton
 ********************************************************************)

(*TODO: Add your comment here*)
FUNCTION_BLOCK Center2

(*Calculate m/min*)
	Calc1:=Speed/0.06;
	(*Calculate Time required for deceleration*)
	DecTime:=Speed/50;
	(*Calculate Distance travelled during deceleration*)
	DecDist:=((Calc1/4)*DecTime);
	(*Calculate Preset TIme for Batch Centering Time Delay*)
	PTReal:=(((Centre-(WidthIn/2))-DecDist)/Calc1)*1000;
	(*Convert real value into UDINT*)
	PT:= REAL_TO_UDINT (PTReal);

END_FUNCTION_BLOCK
```

#### ControlFB.st
```iecst
(* TODO: Add your comment here *)
FUNCTION_BLOCK ControlFB

	//CONTROL CIRCUIT START
	IF(Start)THEN
		BuzzerTON.IN := TRUE;
	END_IF

	//EITHER STOP BUTTON OR STANDBY DELAY DONE SET LATCH
	IF(Stop) OR(StandbyTON.Q)THEN
		StopLatch := TRUE ;
	END_IF

	//WHEN LATCH SET, WAIT FOR LINE EMPTY TO RESET CONTROL READY
	IF(StopLatch) AND(Empty)THEN
		StopDone := TRUE ;
	ELSE
		StopDone := FALSE ;
	END_IF

	//RESET CONDITIONS - ESTOP BUTTONS, TEST MODE, STOP BUTTON OR STANDBY
	IF((EStop1) AND(EStop2)) OR(Test) OR(StopDone)THEN
		BuzzerTON.IN := FALSE ;
		IF NOT(EStopStartTON.IN) THEN
			Achieved1 := FALSE ;
			Achieved2 := FALSE ;
		END_IF
		StopLatch := FALSE ;
		Buzzer := FALSE ;
	ELSE
		IF(EStop1) THEN
			BuzzerTON.IN := FALSE ;
			IF NOT(EStopStartTON.IN) THEN
				Achieved1 := FALSE ;
				Achieved2 := FALSE ;
			END_IF
		END_IF
	END_IF

	//BUZZER WARNING ON CONTROL START AND ALARM
	BuzzerTON.PT := BuzzerPT ;
	BuzzerTON();

	//BUZZER CONTROL AT CONTROL START
	IF EDGEPOS(BuzzerTON.IN)THEN
		Buzzer := TRUE ;
	END_IF

	IF EDGEPOS(BuzzerTON.Q)THEN
		Buzzer := FALSE	;
	END_IF

	//BUZZER CONTROL ON ALARM
	IF EDGEPOS(Alarm)THEN
		Buzzer := TRUE ;
	ELSIF EDGENEG(Alarm)THEN
		Buzzer := FALSE	;
	END_IF

	//BUZZER DISABLE OVERRIDE
	IF (BuzzBlock)THEN
		Buzzer := FALSE	;
	END_IF

	//CONTROL CIRCUITS
	IF(BuzzerTON.Q) THEN
		IF NOT(EStop1)THEN
			Achieved1 := TRUE ;
		END_IF
		IF NOT(EStop2)THEN
			Achieved2 := TRUE ;
		END_IF
	END_IF

	//CONTROL ON LAMPS
	OnLmp1 := Achieved1 ;
	OnLmp2 := Achieved2	;

	//STANDBY DELAY FOR ENERGY SAVING
	IF(Empty) AND(Achieved1) AND(Achieved2) AND NOT(ESClear) AND NOT(StandbyBlock) THEN
		StandbyTON.IN := TRUE ;
	ELSE
		StandbyTON.IN := FALSE	;
	END_IF

	StandbyTON.PT := StandbyPT	;
	StandbyTON ();

	IF EDGEPOS(Stop) OR(StandbyTON.Q)THEN
		StopLatch	:= 	TRUE	;
	END_IF

	//USE CALCULATED NUMBER OF BITS TO DETERMINE WHEN STOP LATCH FINISHES
		FOR i := 0 TO 19 DO
		IF CountIN[i] = TRUE THEN
			Empty := FALSE ;
			EXIT ;
		ELSE
			Empty := TRUE ;
		END_IF
	END_FOR

	//LIGHTSTACK CONTROL
	//GENERATE 1 SEC PULSE FLAG, 0.5 SEC ON, 0.5 SEC OFF.
	TSecON.IN := NOT(TSecOFF.Q)	;
	TSecON.PT := t#500ms ;
	TSecON ();

	TSecOn := TSecON.Q ;
	TSecOFF.IN := TSecOn ;
	TSecOFF.PT := t#500ms ;
	TSecOFF ();

	TSecOff := NOT(TSecOn) ;

	//RED LAMP CONTROL CONDITIONS
	Red[0] := NOT(Achieved1)	;
	Red[1] := (Achieved1) AND(Alarm) AND(TSecOn) ;
	Red[2] := (Achieved1) AND(Warning) AND(TSecOn)	;
	FOR i:= 0 TO 2 DO
		IF (Red[i] = TRUE) THEN
			RedLmp := TRUE ;
			EXIT;
		ELSE
			RedLmp := FALSE ;
		END_IF
	END_FOR

	//YELLOW LAMP CONTROL CONDITIONS
	Yel[0] := (Achieved1) AND(StopLatch) AND(TSecOn) ;
	Yel[1] := (Achieved1) AND(ESClear) ;
	Yel[2] := (Achieved1) AND(Warning) AND(TSecOff) ;
	FOR i:= 0 TO 2 DO
		IF (Yel[i] = TRUE) THEN
			YelLmp := TRUE	;
			EXIT;
		ELSE
			YelLmp := FALSE	;
		END_IF
	END_FOR

	//GREEN LAMP CONTROL CONDITIONS
	Grn[0] := (Achieved1) AND NOT(ESClear) AND NOT(Paused) ;
	Grn[1] := (Achieved1) AND(TSecOff) AND(Paused) ;
	FOR i:= 0 TO 2 DO
		IF (Grn[i] = TRUE) THEN
			GrnLmp := TRUE ;
			EXIT;
		ELSE
			GrnLmp := FALSE	;
		END_IF
	END_FOR

	//ENABLE CONDITIONS FOR TRACKING
	//AT ESTOP LATCH BIT TO ALLOW FOR MOVEMENT OF GLASS ON CONVEYORS AND PALLETS
	IF(EDGEPOS(EStop1))THEN
		EStopStartTON.IN := TRUE ;
	END_IF

	EStopStartTON.PT := T#2s ;
	EStopStartTON ();

	IF EDGEPOS(EStopStartTON.Q)THEN
		EStopStartTON.IN := FALSE ;
	END_IF

	Auto;

END_FUNCTION_BLOCK
```

#### InvTestFB.st
```iecst
(********************************************************************
 * COPYRIGHT --
 ********************************************************************
 * Library: Lib_Ashton
 * File: InvTestFB.st
 * Author: nicke
 ********************************************************************
 * Implementation of library Lib_Ashton
 ********************************************************************)

//InvTest
FUNCTION_BLOCK InvTestFB

	CASE Index OF
		0:	//STOPPED
			Run := FALSE ;
			Rev := FALSE ;
			Speed := AutoSpeedIN ;
		1:	//FORWARD SEAMING SPEED
			Run := TRUE ;
			Rev := FALSE ;
			Speed := SpeedIN.SpeedSeam ;
		2:	//FORWARD TRANSFER SPEED
			Run := TRUE ;
			Rev := FALSE ;
			Speed := SpeedIN.SpeedTrans ;
		3:	//FORWARD MAX SPEED
			Run := TRUE ;
			Rev := FALSE ;
			Speed := SpeedIN.SpeedMax ;
		4:	//FORWARD SLOW SPEED
			Run := TRUE ;
			Rev := FALSE ;
			Speed := SpeedIN.SpeedSlow ;
		5:	//FORWARD LASER SPEED
			Run := TRUE ;
			Rev := FALSE ;
			Speed := SpeedIN.SpeedLaser ;
		6:	//FORWARD WASHER SPEED
			Run := TRUE ;
			Rev := FALSE ;
			Speed := SpeedIN.SpeedWash ;
		7:	//REVERSE SLOW SPEED
			Run := TRUE ;
			Rev := TRUE ;
			Speed := SpeedIN.SpeedSlow ;
		8:	//CENTERING SPEED
			Run := TRUE ;
			Rev := FALSE ;
			Speed :=	SpeedIN.SpeedCntr ;
		9:	//BATCH SPEED
			Run := TRUE ;
			Rev := FALSE ;
			Speed :=	SpeedIN.SpeedBatch ;
		10:	//ENTRY SPEED
			Run := TRUE ;
			Rev := FALSE ;
			Speed :=	SpeedIN.SpeedEntry ;
		11:	//EXIT SPEED
			Run := TRUE ;
			Rev := FALSE ;
			Speed :=	SpeedIN.SpeedExit;
		12: //TEST SPEED FORWARD
			Run := TRUE ;
			Rev := FALSE ;
			Speed := TestSpeedIN ;
		13: //TEST SPEED REVERSE
			Run := TRUE ;
			Rev := TRUE ;
			Speed := TestSpeedIN ;
		14: //TEST ANALOG SPEED
			Run := TRUE ;
			Rev := FALSE ;
			Speed := AnalogSpeedIN ;
		15: //TEST REDUCED SEAMING SPEED
			Run := TRUE ;
			Rev := FALSE ;
			Speed := SpeedIN.SpeedSeamSlow ;
	END_CASE

END_FUNCTION_BLOCK
```

#### SeamersSMProFB.st
```iecst
(* Seamers start up control SMPro *)
FUNCTION_BLOCK SeamersSMProFB

	//ENABLE AUTO START SEQUENCE BUTTON ON SCREEN
	IF(Enable[1]) AND(Enable[2]) AND NOT(AutoStart[1]) AND NOT(AutoStart[2]) THEN
		StartAllDisp := FB_SHOW ;
	ELSE
		StartAllDisp := FB_HIDE ;
	END_IF

	//START AUTO SEQUENCE DURING NORMAL START UP
	IF EDGEPOS(AutoStart[0]) AND NOT(ESClear) THEN
		Latch := TRUE ;
	END_IF

	//START AUTO SEQUENCE AFTER EMO RECOVERY
	IF EDGEPOS(AutoStart[0]) AND(ESClear) AND(ControlIN) THEN
		LatchES := TRUE ;
	END_IF

	//RESET AUTO SEQUENCE BY TURNING OFF ENABLE FOR ALL SEAMERS
	IF NOT(Enable[1]) OR NOT(Enable[2]) THEN
		Latch := FALSE ;
		LatchES := FALSE ;
	END_IF

	//RESET AUTO START
	IF NOT(Enable[1]) THEN
		AutoStart[1] := FALSE ;
	END_IF
	IF NOT(Enable[2]) THEN
		AutoStart[2] := FALSE ;
	END_IF

	//RESET AUTO SEQUENCE AT END OF NORMAL STARTUP
	IF (Vac4TON.Q) AND (Latch) THEN
		Latch := FALSE ;
	END_IF
	//RESET AUTO SEQUENCE AT END OF EMO RESTART
	IF (Vac1TON.Q) AND (LatchES) THEN
		LatchES := FALSE ;
	END_IF

	//-------------------------------------------------------------------------
	//ON CONDITIONS FOR SEAMER 1 AUTO START SEQUENCE
	IF(Enable[1])THEN
		IF (EDGEPOS(Latch)) OR(EDGENEG(Starting2) AND(LatchES)) THEN
			AutoStart[1] := TRUE ;
		END_IF
	END_IF

	IF EDGEPOS(AutoStart[1]) AND NOT(Starting2) THEN
		Starting1 := TRUE ;
	END_IF

	//SEAMER 1 MOTORS AND PUMP START CONTROL
	IF (AutoStart[1]) AND(Enable[1]) AND(ControlIN) THEN
		Belt1TON.IN := TRUE ;
		IF (Extract2TON.Q) THEN
			Starting1 := FALSE ;
		END_IF
	ELSE
		Belt1TON.IN := FALSE ;
		Belt2TON.IN := FALSE ;
		Belt3TON.IN := FALSE ;
		Belt4TON.IN := FALSE ;
		Belt9TON.IN := FALSE ;
		Belt10TON.IN := FALSE ;
		IF NOT(TransportMode) THEN
			Vac1TON.IN := FALSE ;
			Vac2TON.IN := FALSE ;
		END_IF
		ED1TON.IN := FALSE ;
		ED2TON.IN := FALSE ;
		Extract1TON.IN := FALSE ;
		Extract2TON.IN := FALSE ;
		Starting1 := FALSE ;
	END_IF

	//AUTO START SEQUENCE
	Belt1TON.PT := BeltsPT ;
	Belt1TON ();

	Belt2TON.IN := Belt1TON.Q ;
	Belt2TON.PT := BeltsPT ;
	Belt2TON ();

	Belt3TON.IN := Belt2TON.Q ;
	Belt3TON.PT := BeltsPT ;
	Belt3TON ();

	Belt4TON.IN := Belt3TON.Q ;
	Belt4TON.PT := BeltsPT ;
	Belt4TON ();

	Belt9TON.IN := Belt4TON.Q ;
	Belt9TON.PT := BeltsPT ;
	Belt9TON ();

	Belt10TON.IN := Belt9TON.Q ;
	Belt10TON.PT := BeltsPT ;
	Belt10TON ();

	CASE BOOL_TO_INT(TransportMode) OF
		0:
			Vac1TON.IN := Belt9TON.Q ;
		1:
			Vac1TON.IN := TRUE ;
	END_CASE
	Vac1TON.PT := VacPT	;
	Vac1TON ();

	Vac2TON.IN := Vac1TON.Q ;
	Vac2TON.PT := VacPT	;
	Vac2TON ();

	ED1TON.IN := Vac2TON.Q	;
	ED1TON.PT := EDPT	;
	ED1TON ();

	ED2TON.IN := ED1TON.Q	;
	ED2TON.PT := EDPT	;
	ED2TON ();

	Extract1TON.IN := ED2TON.Q	;
	Extract1TON.PT := ExtractionPT	;
	Extract1TON ();

	Extract2TON.IN := Extract1TON.Q	;
	Extract2TON.PT := ExtractionPT	;
	Extract2TON ();

	//OUTPUTS
	IF (Enable[1]) THEN
		BeltOUT[1] := Belt1TON.IN ;
		BeltOUT[2] := Belt2TON.IN ;
		BeltOUT[3] := Belt3TON.IN ;
		BeltOUT[4] := Belt4TON.IN ;
		BeltOUT[9] := Belt9TON.IN ;
		BeltOUT[10] := Belt10TON.IN ;
		VacOUT[1] := Vac1TON.IN OR VacStopTON.IN ;
		VacOUT[2] := Vac2TON.IN OR VacStopTON.IN ;
		EDOUT[1] := ED1TON.IN AND EDOn ;
		EDOUT[2] := ED2TON.IN AND EDOn ;
		ExtractionOUT[1] := Extract1TON.IN ;
		ExtractionOUT[2] := Extract2TON.IN ;
	ELSE
		BeltOUT[1] := FALSE ;
		BeltOUT[2] := FALSE ;
		BeltOUT[3] := FALSE ;
		BeltOUT[4] := FALSE ;
		BeltOUT[9] := FALSE ;
		BeltOUT[10] := FALSE ;
		VacOUT[1] := FALSE ;
		VacOUT[2] := FALSE ;
		EDOUT[1] := FALSE ;
		EDOUT[2] := FALSE ;
		ExtractionOUT[1] := FALSE ;
		ExtractionOUT[2] := FALSE ;
	END_IF

	//AutoStart[1] RESET CONDITIONS
	IF EDGEPOS(AutoStart[1]) AND(Starting2) THEN
		AutoStart[1] := FALSE ;
	END_IF
	IF EDGENEG(AutoStart[1]) OR EDGENEG(Enable[1]) OR NOT(Enable[1]) AND(AutoStart[1]) THEN
		AutoStart[1] := FALSE ;
	END_IF
	IF NOT(ControlIN) OR(Detension) AND(AutoStart[1]) THEN
		AutoStart[1]	:= 	FALSE	;
	END_IF
	IF(AutoStart[1]) THEN
		FOR i:= 1 TO 12 DO
			IF Trips[i] = TRUE THEN
				AutoStart[1]	:= 	FALSE	;
				EXIT				;
			END_IF
		END_FOR
	END_IF

	//DoneOUT[1] CONDITIONS
	IF EDGENEG(Starting1) AND (AutoStart[1]) AND(Enable[1]) THEN
		DoneOUT[1] := TRUE ;
	END_IF
	IF NOT(Starting1) AND NOT(AutoStart[1]) AND(Enable[1]) THEN
		DoneOUT[1] := FALSE ;
	END_IF
	IF NOT(Enable[1]) THEN
		DoneOUT[1] := TRUE ;
	END_IF

	//-------------------------------------------------------------------------
	//ON CONDITIONS FOR SEAMER 2 AUTO START SEQUENCE
	IF(Enable[2])THEN
		IF(EDGENEG(Starting1) AND(Latch)) OR(EDGEPOS(LatchES) AND(Enable[2])) THEN
			AutoStart[2] := TRUE ;
		END_IF
	END_IF

	IF EDGEPOS(AutoStart[2]) AND NOT(Starting1) THEN
		Starting2 := TRUE ;
	END_IF

	//SEAMER 2 MOTORS AND PUMP START CONTROL
	IF (AutoStart[2]) AND(Enable[2]) AND(ControlIN) THEN
		Belt5TON.IN := TRUE ;
		IF (Extract4TON.Q) THEN
			Starting2 := FALSE ;
		END_IF
	ELSE
		Belt5TON.IN := FALSE ;
		Belt6TON.IN := FALSE ;
		Belt7TON.IN := FALSE ;
		Belt8TON.IN := FALSE ;
		Belt11TON.IN := FALSE ;
		Belt12TON.IN := FALSE ;
		IF NOT(TransportMode) THEN
			Vac3TON.IN := FALSE ;
			Vac4TON.IN := FALSE ;
		END_IF
		ED3TON.IN := FALSE ;
		ED4TON.IN := FALSE ;
		Extract3TON.IN := FALSE ;
		Extract4TON.IN := FALSE ;
		Starting2 := FALSE ;
	END_IF

	//AUTO START SEQUENCE
	Belt5TON.PT := BeltsPT ;
	Belt5TON ();

	Belt6TON.IN := Belt5TON.Q ;
	Belt6TON.PT := BeltsPT ;
	Belt6TON ();

	Belt7TON.IN := Belt6TON.Q ;
	Belt7TON.PT := BeltsPT ;
	Belt7TON ();

	Belt8TON.IN := Belt7TON.Q ;
	Belt8TON.PT := BeltsPT ;
	Belt8TON ();

	Belt11TON.IN := Belt8TON.Q ;
	Belt11TON.PT := BeltsPT ;
	Belt11TON ();

	Belt12TON.IN := Belt11TON.Q ;
	Belt12TON.PT := BeltsPT ;
	Belt12TON ();

	CASE BOOL_TO_INT(TransportMode) OF
		0:
			Vac3TON.IN := Belt12TON.Q ;
		1:
			Vac3TON.IN := Vac2TON.Q ;
	END_CASE
	Vac3TON.PT := VacPT	;
	Vac3TON ();

	Vac4TON.IN := Vac3TON.Q ;
	Vac4TON.PT := VacPT	;
	Vac4TON ();

	ED3TON.IN := Vac4TON.Q	;
	ED3TON.PT := EDPT	;
	ED3TON ();

	ED4TON.IN := ED3TON.Q	;
	ED4TON.PT := EDPT	;
	ED4TON ();

	Extract3TON.IN := ED4TON.Q	;
	Extract3TON.PT := ExtractionPT	;
	Extract3TON ();

	Extract4TON.IN := Extract3TON.Q	;
	Extract4TON.PT := ExtractionPT	;
	Extract4TON ();

	//OUTPUTS
	IF (Enable[2]) THEN
		BeltOUT[5] := Belt5TON.IN ;
		BeltOUT[6] := Belt6TON.IN ;
		BeltOUT[7] := Belt7TON.IN ;
		BeltOUT[8] := Belt8TON.IN ;
		BeltOUT[11] := Belt11TON.IN ;
		BeltOUT[12] := Belt12TON.IN ;
		VacOUT[3] := Vac3TON.IN OR VacStopTON.IN ;
		VacOUT[4] := Vac4TON.IN OR VacStopTON.IN ;
		EDOUT[3] := ED3TON.IN AND EDOn ;
		EDOUT[4] := ED4TON.IN AND EDOn ;
		ExtractionOUT[3] := Extract3TON.IN ;
		ExtractionOUT[4] := Extract4TON.IN ;
	ELSE
		BeltOUT[5] := FALSE ;
		BeltOUT[6] := FALSE ;
		BeltOUT[7] := FALSE ;
		BeltOUT[8] := FALSE ;
		BeltOUT[11] := FALSE ;
		BeltOUT[12] := FALSE ;
		VacOUT[3] := FALSE ;
		VacOUT[4] := FALSE ;
		EDOUT[3] := FALSE ;
		EDOUT[4] := FALSE ;
		ExtractionOUT[3] := FALSE ;
		ExtractionOUT[4] := FALSE ;
	END_IF

	//AutoStart[2] RESET CONDITIONS
	IF EDGEPOS(AutoStart[2]) AND(Starting1) AND(AutoStart[2]) THEN
		AutoStart[2] := FALSE ;
	END_IF
	IF EDGENEG(AutoStart[2]) OR EDGENEG(Enable[2]) OR NOT(Enable[2]) AND(AutoStart[2]) THEN
		AutoStart[2] := FALSE ;
	END_IF
	IF NOT(ControlIN) OR(Detension) AND(AutoStart[2]) THEN
		AutoStart[2]	:= 	FALSE	;
	END_IF
	IF(AutoStart[2]) THEN
		FOR i:= 13 TO 24 DO
			IF Trips[i] = TRUE THEN
				AutoStart[2]	:= 	FALSE	;
				EXIT				;
			END_IF
		END_FOR
	END_IF

	//DoneOUT[2] CONDITIONS
	IF EDGENEG(Starting2) AND (AutoStart[2]) AND(Enable[2]) THEN
		DoneOUT[2] := TRUE ;
	END_IF
	IF NOT(Starting2) AND NOT(AutoStart[2]) AND(Enable[2]) THEN
		DoneOUT[2] := FALSE ;
	END_IF
	IF NOT(Enable[2]) THEN
		DoneOUT[2] := TRUE ;
	END_IF

	//-------------------------------------------------------------------------
	//TRANSPORT ONLY MODE - ENABLE VACUUM PUMPS ONLY
	IF(TransportMode) AND(ControlIN) THEN
		VacOUT[1] := TRUE ;
		VacOUT[2] := Vac1TON.Q ;
		VacOUT[3] := Vac2TON.Q ;
		VacOUT[4] := Vac3TON.Q ;
		Enable[1] := FALSE ;
		Enable[2] := FALSE ;
		Enable[3] := FALSE ;
		Enable[4] := FALSE ;
	END_IF

	IF EDGENEG(TransportMode) THEN
		VacOUT[1] := FALSE	;
		VacOUT[2] := FALSE	;
		VacOUT[3] := FALSE	;
		VacOUT[4] := FALSE	;
	END_IF

	//RUN VACUUM PUMPS AFTER CONTROL OFF TO ENSURE DRY AIR PASSING THROUGH
	IF EDGENEG(ControlIN) AND((Enable[1]) OR(Enable[2]) OR(Enable[3]) OR(Enable[4])) THEN
		VacStopTON.IN := TRUE ;
		VacOUT[1] := TRUE ;
		VacOUT[2] := TRUE ;
		VacOUT[3] := TRUE ;
		VacOUT[4] := TRUE ;
	END_IF

	//DELAY BEFORE VACUUM PUMP STOP
	VacStopTON.PT := VacsStopPT ;
	VacStopTON ();

	IF(VacStopTON.Q) THEN
		VacStopTON.IN := FALSE ;
	END_IF

	//WATER CONTROL
	//START CONDITIONS FOR WATER PUMPS
	PumpOUT[1] := FALSE ;
	PumpOUT[2] := FALSE ;
	IF (AutoStart[1]) OR(AutoStart[2]) THEN
		IF(ControlIN) AND NOT(Pump1TON.Q) THEN
			PumpOUT[1] := TRUE ;
		ELSE
			PumpOUT[1] := FALSE ;
		END_IF
		IF (ControlIN) AND NOT(Pump2TON.Q) THEN
			PumpOUT[2] := TRUE ;
		ELSE
			PumpOUT[2] := FALSE ;
		END_IF
	END_IF

	//FLOAT SWITCH CONTROL OF WATER PUMP
	Pump1TON.IN := NOT(Float[1]) ;
	Pump1TON.PT := PumpPT[1] ;
	Pump1TON ();

	Pump2TON.IN := NOT(Float[2]) ;
	Pump2TON.PT := PumpPT[1] ;
	Pump2TON ();

	//SCAVENGE PUMP
	IF (AutoStart[1]) OR(AutoStart[2]) OR(PumpOUT[0]) THEN
		Pump3TON.IN := TRUE ;
	ELSE
		Pump3TON.IN := FALSE ;
	END_IF
	//DELAY BEFORE SCAVENGE PUMP STARTS
	Pump3TON.PT	:= PumpPT[3] ;
	Pump3TON ();

	IF (Pump3TON.Q) AND NOT (Pump4TON.Q) THEN
		PumpOUT[0]	:= 	TRUE	;
	ELSE
		PumpOUT[0]	:= 	FALSE	;
	END_IF

	//DELAY BEFORE SCAVENGE PUMP STOP
	Pump4TON.PT	:= PumpPT[4] ;
	Pump4TON ();

	IF NOT(AutoStart[1]) AND NOT(AutoStart[2]) THEN
		Pump4TON.IN := TRUE ;
	ELSE
		Pump4TON.IN := FALSE ;
	END_IF

END_FUNCTION_BLOCK
```

#### SeamersFB.st
```iecst
(*AUTO START CONTROL OF ALL MOTORS AND PUMPS*)
FUNCTION_BLOCK SeamersFB

	//ENABLE AUTO START SEQUENCE BUTTON ON SCREEN
	IF(Enable[1]) AND(Enable[2]) AND(Enable[3]) AND(Enable[4]) AND NOT(AutoStart[1]) AND NOT(AutoStart[2]) AND NOT(AutoStart[3]) AND NOT(AutoStart[4]) THEN
		StartAllDisp := FB_SHOW ;
	ELSE
		StartAllDisp := FB_HIDE ;
	END_IF

	//START AUTO SEQUENCE DURING NORMAL START UP
	IF EDGEPOS(AutoStart[0]) AND NOT(ESClear) THEN
		Latch := TRUE ;
	END_IF

	//START AUTO SEQUENCE AFTER EMO RECOVERY
	IF EDGEPOS(AutoStart[0]) AND(ESClear) THEN
		LatchES := TRUE ;
	END_IF

	//RESET AUTO SEQUENCE BY TURNING OFF ENABLE FOR ALL SEAMERS
	IF NOT(Enable[1]) OR NOT(Enable[2])  OR NOT(Enable[3]) OR NOT(Enable[4]) THEN
		Latch := FALSE ;
		LatchES := FALSE ;
	END_IF

	//RESET AUTO START
	IF NOT(Enable[1]) THEN
		AutoStart[1] := FALSE ;
	END_IF
	IF NOT(Enable[2]) THEN
		AutoStart[2] := FALSE ;
	END_IF
	IF NOT(Enable[3]) THEN
		AutoStart[3] := FALSE ;
	END_IF
	IF NOT(Enable[4]) THEN
		AutoStart[4] := FALSE ;
	END_IF

	//RESET AUTO SEQUENCE AT END OF NORMAL STARTUP
	IF (Vac4TON.Q) AND (Latch) THEN
		Latch := FALSE ;
	END_IF
	//RESET AUTO SEQUENCE AT END OF EMO RESTART
	IF (Vac1TON.Q) AND (LatchES) THEN
		LatchES := FALSE ;
	END_IF

	//-------------------------------------------------------------------------
	//ON CONDITIONS FOR SEAMER 2 AUTO START SEQUENCE
	IF(Enable[1])THEN
		IF (EDGEPOS(Latch)) OR(EDGENEG(Starting2) AND(LatchES)) THEN
			AutoStart[1] := TRUE ;
		END_IF
	END_IF

	IF EDGEPOS(AutoStart[1]) AND NOT(Starting2) AND NOT(Starting3) AND NOT(Starting4) THEN
		Starting1 := TRUE ;
	END_IF

	//SEAMER 1 MOTORS AND PUMP START CONTROL
	IF (AutoStart[1]) AND(Enable[1]) AND(ControlIN) THEN
		Belt1TON.IN := TRUE ;
		IF (Extract1TON.Q) THEN
			Starting1 := FALSE ;
		END_IF
	ELSE
		Belt1TON.IN := FALSE ;
		Belt2TON.IN := FALSE ;
		Belt9TON.IN := FALSE ;
		IF NOT(TransportMode) THEN
			Vac1TON.IN := FALSE ;
		END_IF
		ED1TON.IN := FALSE ;
		Extract1TON.IN := FALSE ;
		Starting1 := FALSE ;
	END_IF

	//AUTO START SEQUENCE
	Belt1TON.PT := BeltsPT ;
	Belt1TON ();

	Belt2TON.IN := Belt1TON.Q ;
	Belt2TON.PT := BeltsPT ;
	Belt2TON ();

	Belt9TON.IN := Belt2TON.Q ;
	Belt9TON.PT := BeltsPT ;
	Belt9TON ();

	CASE BOOL_TO_INT(TransportMode) OF
		0:
			Vac1TON.IN := Belt9TON.Q ;
		1:
			Vac1TON.IN := TRUE ;
	END_CASE
	Vac1TON.PT := VacPT	;
	Vac1TON ();

	ED1TON.IN := Vac1TON.Q	;
	ED1TON.PT := EDPT	;
	ED1TON ();

	Extract1TON.IN := ED1TON.Q	;
	Extract1TON.PT := ExtractionPT	;
	Extract1TON ();

	//OUTPUTS
	IF (Enable[1]) THEN
		BeltOUT[1] := Belt1TON.IN ;
		BeltOUT[2] := Belt2TON.IN ;
		BeltOUT[9] := Belt9TON.IN ;
		VacOUT[1] := Vac1TON.IN OR VacStopTON.IN ;
		EDOUT[1] := ED1TON.IN AND EDOn ;
		ExtractionOUT[1] := Extract1TON.IN ;
	ELSE
		BeltOUT[1] := FALSE ;
		BeltOUT[2] := FALSE ;
		BeltOUT[9] := FALSE ;
		VacOUT[1] := FALSE ;
		EDOUT[1] := FALSE ;
		ExtractionOUT[1] := FALSE ;
	END_IF

	//AutoStart[1] RESET CONDITIONS
	IF EDGEPOS(AutoStart[1]) AND((Starting2) OR(Starting3) OR(Starting4)) AND(AutoStart[1]) THEN
		AutoStart[1] := FALSE ;
	END_IF
	IF EDGENEG(AutoStart[1]) OR EDGENEG(Enable[1]) OR NOT(Enable[1]) AND(AutoStart[1]) THEN
		AutoStart[1] := FALSE ;
	END_IF
	IF NOT(ControlIN) OR(Detension) AND(AutoStart[1]) THEN
		AutoStart[1]	:= 	FALSE	;
	END_IF
	IF(AutoStart[1]) THEN
		FOR i:= 1 TO 6 DO
			IF Trips[i] = TRUE THEN
				AutoStart[1]	:= 	FALSE	;
				EXIT				;
			END_IF
		END_FOR
	END_IF

	//DoneOUT[1] CONDITIONS
	IF EDGENEG(Starting1) AND (AutoStart[1]) AND(Enable[1]) THEN
		DoneOUT[1] := TRUE ;
	END_IF
	IF NOT(Starting1) AND NOT(AutoStart[1]) AND(Enable[1]) THEN
		DoneOUT[1] := FALSE ;
	END_IF
	IF NOT(Enable[1]) THEN
		DoneOUT[1] := TRUE ;
	END_IF

	//-------------------------------------------------------------------------
	//ON CONDITIONS FOR SEAMER 2 AUTO START SEQUENCE
	IF(Enable[2])THEN
		IF(EDGENEG(Starting1) AND(Latch)) OR(EDGENEG(Starting3) AND(LatchES)) THEN
			AutoStart[2] := TRUE ;
		END_IF
	END_IF

	IF EDGEPOS(AutoStart[2]) AND NOT(Starting1) AND NOT(Starting3) AND NOT(Starting4) THEN
		Starting2 := TRUE ;
	END_IF

	//SEAMER 2 MOTORS AND PUMP START CONTROL
	IF (AutoStart[2]) AND(Enable[2]) AND(ControlIN) THEN
		Belt3TON.IN := TRUE ;
		IF (Extract2TON.Q) THEN
			Starting2 := FALSE ;
		END_IF
	ELSE
		Belt3TON.IN := FALSE ;
		Belt4TON.IN := FALSE ;
		Belt10TON.IN := FALSE ;
		IF NOT(TransportMode) THEN
			Vac2TON.IN := FALSE ;
		END_IF
		ED2TON.IN := FALSE ;
		Extract2TON.IN := FALSE ;
		Starting2 := FALSE ;
	END_IF

	//AUTO START SEQUENCE
	Belt3TON.PT := BeltsPT ;
	Belt3TON ();

	Belt4TON.IN := Belt3TON.Q ;
	Belt4TON.PT := BeltsPT ;
	Belt4TON ();

	Belt10TON.IN := Belt4TON.Q ;
	Belt10TON.PT := BeltsPT ;
	Belt10TON ();

	CASE BOOL_TO_INT(TransportMode) OF
		0:
			Vac2TON.IN := Belt10TON.Q ;
		1:
			Vac2TON.IN := Vac1TON.Q ;
	END_CASE
	Vac2TON.PT := VacPT	;
	Vac2TON ();

	ED2TON.IN := Vac2TON.Q	;
	ED2TON.PT := EDPT	;
	ED2TON ();

	Extract2TON.IN := ED2TON.Q	;
	Extract2TON.PT := ExtractionPT	;
	Extract2TON ();

	//OUTPUTS
	IF (Enable[2]) THEN
		BeltOUT[3] := Belt3TON.IN ;
		BeltOUT[4] := Belt4TON.IN ;
		BeltOUT[10] := Belt10TON.IN ;
		VacOUT[2] := Vac2TON.IN OR VacStopTON.IN ;
		EDOUT[2] := ED2TON.IN AND EDOn ;
		ExtractionOUT[2] := Extract2TON.IN ;
	ELSE
		BeltOUT[3] := FALSE ;
		BeltOUT[4] := FALSE ;
		BeltOUT[10] := FALSE ;
		VacOUT[2] := FALSE ;
		EDOUT[2] := FALSE ;
		ExtractionOUT[2] := FALSE ;
	END_IF

	//AutoStart[2] RESET CONDITIONS
	IF EDGEPOS(AutoStart[2]) AND((Starting1) OR(Starting3) OR(Starting4)) AND(AutoStart[2]) THEN
		AutoStart[2] := FALSE ;
	END_IF
	IF EDGENEG(AutoStart[2]) OR EDGENEG(Enable[2]) OR NOT(Enable[2]) AND(AutoStart[2]) THEN
		AutoStart[2] := FALSE ;
	END_IF
	IF NOT(ControlIN) OR(Detension) AND(AutoStart[2]) THEN
		AutoStart[2]	:= 	FALSE	;
	END_IF
	IF(AutoStart[2]) THEN
		FOR i:= 7 TO 12 DO
			IF Trips[i] = TRUE THEN
				AutoStart[2]	:= 	FALSE	;
				EXIT				;
			END_IF
		END_FOR
	END_IF

	//DoneOUT[2] CONDITIONS
	IF EDGENEG(Starting2) AND (AutoStart[2]) AND(Enable[2]) THEN
		DoneOUT[2] := TRUE ;
	END_IF
	IF NOT(Starting2) AND NOT(AutoStart[2]) AND(Enable[2]) THEN
		DoneOUT[2] := FALSE ;
	END_IF
	IF NOT(Enable[2]) THEN
		DoneOUT[2] := TRUE ;
	END_IF

	//-------------------------------------------------------------------------
	//ON CONDITIONS FOR SEAMER 3 AUTO START SEQUENCE
	IF(Enable[3])THEN
		IF(EDGENEG(Starting2) AND(Latch)) OR(EDGENEG(Starting4) AND(LatchES)) THEN
			AutoStart[3] := TRUE ;
		END_IF
	END_IF

	IF EDGEPOS(AutoStart[3]) AND NOT(Starting1) AND NOT(Starting2) AND NOT(Starting4) THEN
		Starting3 := TRUE ;
	END_IF

	//SEAMER 3 MOTORS AND PUMP START CONTROL
	IF (AutoStart[3]) AND(Enable[3]) AND(ControlIN) THEN
		Belt5TON.IN := TRUE ;
		IF (Extract3TON.Q) THEN
			Starting3 := FALSE ;
		END_IF
	ELSE
		Belt5TON.IN := FALSE ;
		Belt6TON.IN := FALSE ;
		Belt11TON.IN := FALSE ;
		IF NOT(TransportMode) THEN
			Vac3TON.IN := FALSE ;
		END_IF
		ED3TON.IN := FALSE ;
		Extract3TON.IN := FALSE ;
		Starting3 := FALSE ;
	END_IF

	//AUTO START SEQUENCE
	Belt5TON.PT := BeltsPT ;
	Belt5TON ();

	Belt6TON.IN := Belt5TON.Q ;
	Belt6TON.PT := BeltsPT ;
	Belt6TON ();

	Belt11TON.IN := Belt6TON.Q ;
	Belt11TON.PT := BeltsPT ;
	Belt11TON ();

	CASE BOOL_TO_INT(TransportMode) OF
		0:
			Vac3TON.IN := Belt11TON.Q ;
		1:
			Vac3TON.IN := Vac2TON.Q ;
	END_CASE
	Vac3TON.PT := VacPT	;
	Vac3TON ();

	ED3TON.IN := Vac3TON.Q	;
	ED3TON.PT := EDPT	;
	ED3TON ();

	Extract3TON.IN := ED3TON.Q	;
	Extract3TON.PT := ExtractionPT	;
	Extract3TON ();

	//OUTPUTS
	IF (Enable[3]) THEN
		BeltOUT[5] := Belt5TON.IN ;
		BeltOUT[6] := Belt6TON.IN ;
		BeltOUT[11] := Belt11TON.IN ;
		VacOUT[3] := Vac3TON.IN OR VacStopTON.IN ;
		EDOUT[3] := ED3TON.IN AND EDOn ;
		ExtractionOUT[3] := Extract3TON.IN ;
	ELSE
		BeltOUT[5] := FALSE ;
		BeltOUT[6] := FALSE ;
		BeltOUT[11] := FALSE ;
		VacOUT[3] := FALSE ;
		EDOUT[3] := FALSE ;
		ExtractionOUT[3] := FALSE ;
	END_IF

	//AutoStart[3] RESET CONDITIONS
	IF EDGEPOS(AutoStart[3]) AND((Starting1) OR(Starting2) OR(Starting4)) AND(AutoStart[3]) THEN
		AutoStart[3] := FALSE ;
	END_IF
	IF EDGENEG(AutoStart[3]) OR EDGENEG(Enable[3]) OR NOT(Enable[3]) AND(AutoStart[3]) THEN
		AutoStart[3] := FALSE ;
	END_IF
	IF NOT(ControlIN) OR(Detension) AND(AutoStart[3]) THEN
		AutoStart[3]	:= 	FALSE	;
	END_IF
	IF(AutoStart[3]) THEN
		FOR i:= 13 TO 18 DO
			IF Trips[i] = TRUE THEN
				AutoStart[3]	:= 	FALSE	;
				EXIT				;
			END_IF
		END_FOR
	END_IF

	//DoneOUT[3] CONDITIONS
	IF EDGENEG(Starting3) AND (AutoStart[3]) AND(Enable[3]) THEN
		DoneOUT[3] := TRUE ;
	END_IF
	IF NOT(Starting3) AND NOT(AutoStart[3]) AND(Enable[3]) THEN
		DoneOUT[3] := FALSE ;
	END_IF
	IF NOT(Enable[3]) THEN
		DoneOUT[3] := TRUE ;
	END_IF

	//-------------------------------------------------------------------------
	//ON CONDITIONS FOR SEAMER 4 AUTO START SEQUENCE
	IF(Enable[4])THEN
		IF (EDGENEG(Starting3) AND(Latch)) OR(EDGEPOS(LatchES)) THEN
			AutoStart[4] := TRUE ;
		END_IF
	END_IF

	IF EDGEPOS(AutoStart[4]) AND NOT(Starting1) AND NOT(Starting2) AND NOT(Starting3) THEN
		Starting4 := TRUE ;
	END_IF

	//SEAMER 4 MOTORS AND PUMP START CONTROL
	IF (AutoStart[4]) AND(Enable[4]) AND(ControlIN) THEN
		Belt7TON.IN := TRUE ;
		IF (Extract4TON.Q) THEN
			Starting4 := FALSE ;
		END_IF
	ELSE
		Belt7TON.IN := FALSE ;
		Belt8TON.IN := FALSE ;
		Belt12TON.IN := FALSE ;
		IF NOT(TransportMode) THEN
			Vac4TON.IN := FALSE ;
		END_IF
		ED4TON.IN := FALSE ;
		Extract4TON.IN := FALSE ;
		Starting4 := FALSE ;
	END_IF

	//AUTO START SEQUENCE
	Belt7TON.PT := BeltsPT ;
	Belt7TON ();

	Belt8TON.IN := Belt7TON.Q ;
	Belt8TON.PT := BeltsPT ;
	Belt8TON ();

	Belt12TON.IN := Belt8TON.Q ;
	Belt12TON.PT := BeltsPT ;
	Belt12TON ();

	CASE BOOL_TO_INT(TransportMode) OF
		0:
			Vac4TON.IN := Belt12TON.Q ;
		1:
			Vac4TON.IN := Vac3TON.IN ;
	END_CASE
	Vac4TON.PT := VacPT	;
	Vac4TON ();

	ED4TON.IN := Vac4TON.Q	;
	ED4TON.PT := EDPT	;
	ED4TON ();

	Extract4TON.IN := ED4TON.Q	;
	Extract4TON.PT := ExtractionPT	;
	Extract4TON ();

	//OUTPUTS
	IF (Enable[4]) THEN
		BeltOUT[7] := Belt7TON.IN ;
		BeltOUT[8] := Belt8TON.IN ;
		BeltOUT[12] := Belt12TON.IN ;
		VacOUT[4] := Vac4TON.IN OR VacStopTON.IN ;
		EDOUT[4] := ED4TON.IN AND EDOn ;
		ExtractionOUT[4] := Extract4TON.IN ;
	ELSE
		BeltOUT[7] := FALSE ;
		BeltOUT[8] := FALSE ;
		BeltOUT[12] := FALSE ;
		VacOUT[4] := FALSE ;
		EDOUT[4] := FALSE ;
		ExtractionOUT[4] := FALSE ;
	END_IF

	//AutoStart[4] RESET CONDITIONS
	IF EDGEPOS(AutoStart[4]) AND((Starting1) OR(Starting2) OR(Starting3)) AND(AutoStart[4]) THEN
		AutoStart[4] := FALSE ;
	END_IF
	IF EDGENEG(AutoStart[4]) OR EDGENEG(Enable[4]) OR NOT(Enable[4]) AND(AutoStart[4]) THEN
		AutoStart[4] := FALSE ;
	END_IF
	IF NOT(ControlIN) OR(Detension) AND(AutoStart[4]) THEN
		AutoStart[4]	:= 	FALSE	;
	END_IF
	IF(AutoStart[4]) THEN
		FOR i:= 19 TO 24 DO
			IF Trips[i] = TRUE THEN
				AutoStart[4]	:= 	FALSE	;
				EXIT				;
			END_IF
		END_FOR
	END_IF

	//DoneOUT[4] CONDITIONS
	IF EDGENEG(Starting4) AND (AutoStart[4]) AND(Enable[4]) THEN
		DoneOUT[4] := TRUE ;
	END_IF
	IF NOT(Starting4) AND NOT(AutoStart[4]) AND(Enable[4]) THEN
		DoneOUT[4] := FALSE ;
	END_IF
	IF NOT(Enable[4]) THEN
		DoneOUT[4] := TRUE ;
	END_IF

	//-------------------------------------------------------------------------
	//TRANSPORT ONLY MODE - ENABLE VACUUM PUMPS ONLY
	IF(TransportMode) AND(ControlIN) THEN
		VacOUT[1] := TRUE ;
		VacOUT[2] := Vac1TON.Q ;
		VacOUT[3] := Vac2TON.Q ;
		VacOUT[4] := Vac3TON.Q ;
		Enable[1] := FALSE ;
		Enable[2] := FALSE ;
		Enable[3] := FALSE ;
		Enable[4] := FALSE ;
	END_IF

	IF EDGENEG(TransportMode) THEN
		VacOUT[1] := FALSE	;
		VacOUT[2] := FALSE	;
		VacOUT[3] := FALSE	;
		VacOUT[4] := FALSE	;
	END_IF

	//RUN VACUUM PUMPS AFTER CONTROL OFF TO ENSURE DRY AIR PASSING THROUGH
	IF EDGENEG(ControlIN) AND((Enable[1]) OR(Enable[2]) OR(Enable[3]) OR(Enable[4])) THEN
		VacStopTON.IN := TRUE ;
		VacOUT[1] := TRUE ;
		VacOUT[2] := TRUE ;
		VacOUT[3] := TRUE ;
		VacOUT[4] := TRUE ;
	END_IF

	//DELAY BEFORE VACUUM PUMP STOP
	VacStopTON.PT := VacsStopPT ;
	VacStopTON ();

	IF(VacStopTON.Q) THEN
		VacStopTON.IN := FALSE ;
	END_IF

	//WATER CONTROL
	//START CONDITIONS FOR WATER PUMPS
	IF (AutoStart[1]) OR(AutoStart[2]) OR(AutoStart[3]) OR(AutoStart[4]) OR(PumpOUT[1]) THEN
		IF(ControlIN) AND NOT(Pump1TON.Q) THEN
			PumpOUT[1] := TRUE ;
		ELSE
			PumpOUT[1] := FALSE ;
		END_IF
	ELSE
		IF (ControlIN) AND NOT(Pump2TON.Q) THEN
			PumpOUT[2] := TRUE ;
		ELSE
			PumpOUT[2] := FALSE ;
		END_IF
	END_IF

	//FLOAT SWITCH CONTROL OF WATER PUMP
	Pump1TON.IN := NOT(Float[1]) ;
	Pump1TON.PT := PumpPT[1] ;
	Pump1TON ();

	Pump2TON.IN := NOT(Float[2]) ;
	Pump2TON.PT := PumpPT[1] ;
	Pump2TON ();

	//SCAVENGE PUMP
	IF (AutoStart[1]) OR(AutoStart[2]) OR(AutoStart[3]) OR(AutoStart[4]) OR(PumpOUT[0]) THEN
		Pump3TON.IN := TRUE ;
	ELSE
		Pump3TON.IN := FALSE ;
	END_IF
	//DELAY BEFORE SCAVENGE PUMP STARTS
	Pump3TON.PT	:= PumpPT[3] ;
	Pump3TON ();

	IF (Pump3TON.Q) AND NOT (Pump4TON.Q) THEN
		PumpOUT[0]	:= 	TRUE	;
	ELSE
		PumpOUT[0]	:= 	FALSE	;
	END_IF

	//DELAY BEFORE SCAVENGE PUMP STOP
	Pump4TON.PT	:= PumpPT[4] ;
	Pump4TON ();

	IF NOT(AutoStart[1]) OR(AutoStart[2]) OR(AutoStart[3]) OR(AutoStart[4]) THEN
		Pump4TON.IN := TRUE ;
	ELSE
		Pump4TON.IN := FALSE ;
	END_IF

END_FUNCTION_BLOCK
```

#### TrackBit.st
```iecst
(********************************************************************
 * COPYRIGHT --
 ********************************************************************
 * Library: Ashton
 * File: TrackBit.st
 * Author: nicke
 ********************************************************************)

//TRACKING BIT CONTROLS
FUNCTION_BLOCK TrackBit

	//VISUALISATION DISPLAY CONTROLS 0=SHOW, 1 =HIDE
	Disp	:=	FB_SHOW	;
	IF(FixedIN.ESClearing) THEN
		ESDisp	:=	FB_SHOW	;
	ELSE
		ESDisp	:=	FB_HIDE	;
	END_IF

	//OUTPUT CONDITIONS
	Active	:=	TRUE	;
	IF NOT((RunBlock) OR(TimeoutOUT))  THEN
		RunOUT	:=	TRUE	;
		CASE Analog OF
			0:
				SpeedOUT	:=	Speed	;
				IF(SpeedMatchEN) THEN
					SpeedOUT	:=	SpeedMatch	;
				END_IF
			ELSE
				SpeedOUT	:=	SpeedAnalog	;
		END_CASE
	ELSE
		RunOUT	:=	FALSE	;
		SpeedOUT	:=	0.0	;
	END_IF
	IF NOT(SolBlock) THEN
		SolOUT	:=	TRUE	;
	ELSE
		SolOUT	:=	FALSE	;
	END_IF

	//DELAYS
	DelayTON.PT	:= 	DelayPT	;
	DelayTON ();
	//TRACK DELAY
	IF(FixedIN.Control) AND NOT(FixedIN.ESClear) THEN
		IF(TrackDelayEN) THEN
			IF NOT(RunBlock) THEN
				DelayTON.IN	:= 	TRUE	;
			ELSE
				DelayTON.IN	:=	FALSE	;
			END_IF
			IF(DelayTON.Q) THEN
				Done	:=	TRUE	;
			END_IF
		END_IF
	END_IF

	//TIMEOUT CONDITIONS
	IF(FixedIN.Control) THEN
		IF(TimeoutEN) AND NOT(FixedIN.ESClear) THEN
			IF NOT((TimeoutBlock) OR(RunBlock) OR(SolBlock)) THEN
				DelayTON.IN	:= 	TRUE	;

				TimeoutOUT	:= 	DelayTON.Q	;
				IF(TimeoutACK) OR(TimeoutACKLatch) THEN
					TimeoutOUT	:=	FALSE	;
					TimeoutACKLatch	:=	TRUE	;
				END_IF
			ELSE
				TimeoutOUT	:=	FALSE	;
			END_IF
		ELSE
			TimeoutOUT	:=	FALSE	;
		END_IF
	END_IF

	IF(TimeoutOUT) THEN
		RunOUT := FALSE	;
	END_IF

	//DONE CONDITIONS
	IF(DoneIN) AND((FixedIN.Control) OR(FixedIN.EMOStart)) AND NOT(FixedIN.ESClear)  THEN
		Done := TRUE ;
	END_IF

	IF NOT(FixedIN.Control) THEN
		RunOUT := FALSE ;
		TimeoutOUT	:=	FALSE	;
	END_IF

END_FUNCTION_BLOCK
```

#### TrackingSection.st
```iecst
(********************************************************************
 * COPYRIGHT --
 ********************************************************************
 * Library: Ashton
 * File: TrackingSection.st
 * Author: nicke
 ********************************************************************)

//TRACKING SECTION CONTROLS
FUNCTION_BLOCK TrackingSection

	//INDEX FOR TRACKBITS CONTROL
	Index	:=	IndexIN	;

	IF(Index > 0) THEN
		//VISUALISATION DISPLAY CONTROLS
		BusyDisp	:=	FB_SHOW	;
		//OUTPUT CONDITIONS
		Busy	:=	TRUE	;
	ELSE
		BusyDisp	:= 	FB_HIDE	;
		Busy	:=	FALSE	;
	END_IF
	//HIDE DURING ESTOP RECOVERY
	IF(ESDispInhib) THEN
		BusyDisp	:= 	FB_HIDE	;
	END_IF

	IF(Busy) THEN
		//CHECK ARRAY FOR ON CONDITIONS
		IF NOT(BlockInhib) THEN
			FOR i:= 0 TO 12 DO
				IF Blocks[i] = TRUE THEN
					Blocked	:= 	TRUE	;
					EXIT;
				ELSE
					IF NOT(ControlIN) THEN
						Blocked	:= 	TRUE	;
					ELSE
						Blocked	:= 	FALSE	;
					END_IF
				END_IF
			END_FOR
		ELSE
			Blocked	:=	FALSE	;
		END_IF

		//DATA FOR TRANSFER TO NEXT SECTION
		Width	:=	WidthIN	;
		Length	:=	LengthIN	;
		Longest	:=	LongestIN	;
		RowBlock	:=	RowBlockIN	;
		Change	:=	ChangeIN	;
		ArrissUpper	:=	ArrissUpperIN	;
		ArrissLower	:=	ArrissLowerIN	;
		EdgeDelete	:=	EdgeDeleteIN	;
		VerticalBelt	:=	VerticalBeltIN	;
		BatchClear := BatchClearIN ;
		//FIXED VALUES WHILE BUSY
		FixedOUT.Control	:=	ControlIN	;
		FixedOUT.ESClearing	:=	Cleared	;
		FixedOUT.EMOStart := EMOStart ;
		FixedOUT.ESClear := ESClear ;

		//RESET CONDITIONS FROM MIMIC (> OPERATOR LEVEL) OR ESTOP RECOVERY
		IF(ResMan) OR(ResES) THEN
			IndexIN	:= 0 ;
			Index := 0 ;
			WidthIN	:= 0.0	;
			Width := 0.0 ;
			LengthIN :=	0.0	;
			Length := 0.0 ;
			LongestIN := 0.0 ;
			Longest := 0.0 ;
			RowBlockIN := FALSE ;
			ChangeIN :=	FALSE ;
			ArrissUpperIN := FALSE ;
			ArrissLowerIN := FALSE ;
			EdgeDeleteIN :=	FALSE ;
			VerticalBeltIN := FALSE	;
			BatchClearIN := FALSE ;
			BatchClear := FALSE ;
		END_IF
	ELSE
		WidthIN	:=	0.0	;
		Width := 0.0 ;
		LengthIN :=	0.0	;
		Length := 0.0 ;
		LongestIN := 0.0 ;
		Longest := 0.0 ;
		RowBlockIN :=	FALSE	;
		ChangeIN :=	FALSE	;
		ArrissUpperIN	:=	FALSE	;
		ArrissLowerIN	:=	FALSE	;
		EdgeDeleteIN	:=	FALSE	;
		VerticalBeltIN	:=	FALSE	;
		BatchClearIN := FALSE ;
		BatchClear := FALSE ;
		Blocked	:=	FALSE	;
		FixedOUT.Control	:=	FALSE	;
		FixedOUT.ESClearing	:=	FALSE	;
		FixedOUT.ESClear := FALSE ;
	END_IF

	IF EDGEPOS(Busy) THEN
		PreviousTime	:=	CurrentTime	;
		CurrentTime		:=	clock_ms()	;
		ElapsedTime		:=	TIME_TO_UDINT(CurrentTime - PreviousTime)	;
	END_IF

	Cycle	:=	UDINT_TO_REAL(ElapsedTime/1000)	;

END_FUNCTION_BLOCK
```

#### Lib_Ashton.typ
```iecst
TYPE
	IntervalDelays_typ : 	STRUCT
		IntervalPT : UDINT;
		OpenPT : UDINT;
	END_STRUCT;
	IntervalOpen_enum :
		(
		IO_IDLE,
		IO_INTERVAL,
		IO_OPEN
		);
	CycleTime_typ : 	STRUCT
		Current : TIME; (*Current captured time*)
		Previous : TIME; (*Previous captured time*)
		Elapsed : UDINT; (*Elapsed/Cycle time*)
	END_STRUCT;
	Display_enum :
		(
		FB_SHOW := 0,
		FB_HIDE := 1
		);
	TrackBit_Fixed_typ : 	STRUCT
		Control : BOOL;
		ESClearing : BOOL;
		ESClear : BOOL;
		EMOStart : BOOL;
	END_STRUCT;
	FB_ANALOG_enum :
		(
		NO_ANALOG := 0, (*ANALOG NOT SELECTED*)
		VOLTAGE_TYPE_1 := 1, (*0-10V Voltage Type*)
		CURRENT_TYPE_1 := 2, (*0-20mA Current Type*)
		CURRENT_TYPE_2 := 3 (*4-20mA Current Type*)
		);
	PLInvPerm : 	STRUCT
		SpeedMax : REAL; (*Maximum Speed*)
		SpeedSeam : REAL; (*Seaming Speed*)
		SpeedTrans : REAL; (*Transfer Speed*)
		SpeedSlow : REAL; (*Squaring speed*)
		SpeedLaser : REAL; (*Positioning Speed E.G. Laser*)
		SpeedWash : REAL; (*Washer Speed*)
		SpeedCntr : REAL; (*Centering Speed*)
		SpeedBatch : REAL; (*Batching Speed*)
		SpeedEntry : REAL; (*Entry Speed - to match other equipment*)
		SpeedExit : REAL; (*Exit Speed - to match other equipment*)
		SpeedSeamSlow : REAL; (*Slow Seaming Speed*)
	END_STRUCT;
	BATCHTYPE_enum :
		(
		ROW := 0, (*Row Builidng*)
		LOAD := 1 (*Load Building*)
		);
	BATCHING_enum :
		(
		AUTO := 0, (*Auto Batching, to max limits*)
		SINGLE := 1, (*Batching only single pieces*)
		PAIRS := 2, (*Batching only 1 row of 2 pieces*)
		TWOS := 3, (*Batching only 2 rows of 1 piece/row*)
		FOURS := 4 (*Batching only 2 rows of 2 pieces*)
		);
	NozzleControl_enum :
		(
		NC_Idle,
		NC_Open,
		NC_Close,
		NC_CleanDone,
		NC_ControlStop1,
		NC_ControlStop2
		);
	NozzleControl_typ : 	STRUCT
		CountPurge : INT;
		Seq : NozzleControl_enum;
		PurgeCount : INT;
		Delay : INT;
		VacuumStopDelay : DINT;
		NozzleOpenDelay : DINT;
	END_STRUCT;
	NozzlePerm_typ : 	STRUCT
		PurgeCount : INT;
		OpenDelay : DINT;
	END_STRUCT;
	Preset_Seamers_typ : 	STRUCT
		Belt : UDINT; (*During Belt auto start*)
		Vac : UDINT; (*During Vacuum auto start*)
		ED : UDINT; (*During ED auto start*)
		Extraction : UDINT; (*During Extraction auto start*)
		VacsStop : UDINT; (*Vacuum run on after control stop*)
		Water : ARRAY[0..4]OF UDINT; (*Water Pump delays*)
	END_STRUCT;
	Control_typ : 	STRUCT
		Achieved : BOOL;
		ESClear : BOOL;
	END_STRUCT;
	Interval_typ : 	STRUCT
		Out : BOOL; (*Valve output*)
		Open : TON; (*Valve open delay*)
		Interval : TON; (*Interval delay*)
		TestIndex2 : USINT;
		TestIndex1 : USINT;
		FreqIndex : USINT;
	END_STRUCT;
	SeamerStart_enum :
		(
		SS_Reset := 0,
		SS_Ready := 1,
		SS_BeltMotor1 := 2, (*Control for 1st belt motor*)
		SS_BeltMotor2 := 3, (*Control for 2nd belt motor*)
		SS_BeltMotor3 := 4, (*Control for 3rd belt motor*)
		SS_BeltMotor4 := 5, (*Control for 4th belt motor*)
		SS_BeltMotor5 := 6, (*Control for 5th belt motor (Vertical)*)
		SS_BeltMotor6 := 7, (*Control for 6th belt motor (Vertical)*)
		SS_VacuumPump1 := 8, (*Control for 1st vacuum pump*)
		SS_VacuumPump2 := 9, (*Control for 2nd vacuum pump*)
		SS_Extraction1 := 10, (*Control for 1st extraction pump (Dry)*)
		SS_Extraction2 := 11, (*Control for 2nd extraction pump (Dry)*)
		SS_Started := 12,
		SS_TransportMode := 13
		);
	Control_BackGround_typ : 	STRUCT
		Achieved1 : BOOL;
		Achieved2 : BOOL;
		ESClear : BOOL;
		Warning : BOOL;
		Alarm : BOOL;
		AutoStart : ARRAY[0..2]OF BOOL;
		Enable : ARRAY[0..2]OF BOOL;
		ED : BOOL;
	END_STRUCT;
	VacuumRunOn_enum :
		(
		VR_Idle := 0,
		VR_Running := 1,
		VR_Done := 2
		);
	IntervalDelay_enum :
		(
		ID_Idle := 0,
		ID_Interval := 1,
		ID_Open := 2
		);
END_TYPE
```

#### Batch.st
```iecst
//ROW BUILDING CALCULATIONS
FUNCTION_BLOCK Batch

	//RESET
	Done := FALSE ;

	//CAPTURE NEXT WIDTH TO ADD TO ROW
	IF(FollowingIN[0] > 0)THEN
		NextINT := FollowingIN[0] ;
	END_IF

	//PERFORM CALCULATION AS GLASS ARRIVES
	IF EDGENEG(Calculate) AND(Current > 0) THEN
		Current := Current + NextINT + Gap ;
		NextINT := 0 ;
	END_IF

	IF EDGENEG(Calculate) AND(Current = 0) THEN
		Current := NextINT ;
		NextINT := 0 ;
	END_IF

	//CALCULATE COMBINED SIZE WITH FOLLOWING PIECE. IF NO PIECE WAIT UNTIL MEASURED.
	FOR i := 0 TO 9 DO
		IF(FollowingIN[i] > 0) THEN
			Next := FollowingIN[i] ;
			EXIT;
		ELSE
			Next := 0 ;
		END_IF
	END_FOR

	//CALCULATE WHEN COMPLETE
	CASE Type OF
		ROW:
			MinRemaining :=  Gap + 150.0 ;
		LOAD:
			MinRemaining :=  Gap + 300.0 ;
	END_CASE
	CASE BatchMode OF
		AUTO:
			IF(Building) THEN
				NextSize := Current + Next + Gap ;
				Remaining	:=	MaxSize - Current ;
				IF(MinRemaining > Remaining) OR(NextSize > MaxSize) THEN
					Done := TRUE ;
				END_IF
			END_IF
		SINGLE:
			IF(Building) THEN
				Done := TRUE ;
			END_IF
		TWOS:
			CASE Type OF
				ROW:
					IF(Building) THEN
						Done := TRUE ;
					END_IF
				LOAD:
					IF NOT(Building) THEN
						DoubleCount := 0 ;
					END_IF
					IF(Building) THEN
						NextSize := Current + Next + Gap ;
						Remaining	:=	MaxSize - Current ;
						IF(MinRemaining > Remaining) OR(NextSize > MaxSize) THEN
							Done := TRUE ;
							DoubleCount := 2 ;
						END_IF
					END_IF
					IF EDGENEG(Calculate) AND(DoubleCount=1) THEN
						DoubleCount := 2 ;
					END_IF
					IF EDGENEG(Calculate) AND(DoubleCount=0) THEN
						DoubleCount := 1 ;
					END_IF
					IF(DoubleCount=2) THEN
						Done := TRUE ;
					END_IF
			END_CASE
		PAIRS:
			CASE Type OF
				ROW:
					IF NOT(Building) THEN
						DoubleCount := 0 ;
					END_IF
					IF(Building) THEN
						NextSize := Current + Next + Gap ;
						Remaining	:=	MaxSize - Current ;
						IF(MinRemaining > Remaining) OR(NextSize > MaxSize) THEN
							Done := TRUE ;
							DoubleCount := 2 ;
						END_IF
					END_IF
					IF EDGENEG(Calculate) AND(DoubleCount=1) THEN
						DoubleCount := 2 ;
					END_IF
					IF EDGENEG(Calculate) AND(DoubleCount=0) THEN
						DoubleCount := 1 ;
					END_IF
					IF(DoubleCount=2) THEN
						Done := TRUE ;
					END_IF
				LOAD:
					IF(Building) THEN
						Done := TRUE ;
					END_IF
			END_CASE
		FOURS:
			IF NOT(Building) THEN
				DoubleCount := 0 ;
			END_IF
			IF(Building) THEN
				NextSize := Current + Next + Gap ;
				Remaining	:=	MaxSize - Current ;
				IF(MinRemaining > Remaining) OR(NextSize > MaxSize) THEN
					Done := TRUE ;
					DoubleCount := 2 ;
				END_IF
			END_IF
			IF EDGENEG(Calculate) AND(DoubleCount=1) THEN
				DoubleCount := 2 ;
			END_IF
			IF EDGENEG(Calculate) AND(DoubleCount=0) THEN
				DoubleCount := 1 ;
			END_IF
			IF(DoubleCount=2) THEN
				Done := TRUE ;
			END_IF
	END_CASE

	//RESET WHEN NOT ROW BUILDING
	IF NOT(Building) THEN
		Current := 0.0 ;
		Longest := 0.0 ;
		Remaining := MaxSize ;
	END_IF

	IF EDGEPOS(ClearIN) THEN
		Done := TRUE ;
	END_IF

	//CAPTURE NEXT LENGTH
	IF(LengthIN > 0)THEN
		NextLengthINT := LengthIN ;
	END_IF

	//CALCULATE LONGEST IN ROW
	IF EDGENEG(Calculate) AND(NextLengthINT>=0) THEN
		IF(NextLengthINT > Longest) THEN
			Longest := NextLengthINT ;
		END_IF
		NextLengthINT := 0 ;
	END_IF

	//CALCULATE CENTERING TIME
	Center.WidthIn := Current ;
	Center.Speed := CenterSpeed	 ;
	Center.Centre := CenterDist ;
	Center ();
	CenterPT := (Center.PT * 10) ;

END_FUNCTION_BLOCK
```

#### FlipUps.st
```iecst
//FLIP UP ARMS CONTROL
FUNCTION_BLOCK FlipUps

	//CHECK ALL ARMS ARE DOWN BEFORE SEEK AND FIND
	DownDone := FALSE ;

	FOR i := 1 TO (USINT_TO_INT(Arms * 2)) DO
		IF NOT(Down[i]) THEN
			EXIT ;
		ELSIF (i = (USINT_TO_INT(Arms) * 2)) THEN
			DownDone := TRUE ;
		END_IF
	END_FOR

	IF EDGEPOS(Raise) AND NOT(HiVol) THEN
		FOR i := Arms TO 0 BY -1 DO
			IF (ActPos > ArmPos[i]) THEN
				CheckRaised := INT_TO_USINT(i) ;
				EXIT ;
			END_IF
		END_FOR
	END_IF

	IF(HiVol) THEN
		FOR i := Arms TO 0 BY -1 DO
			IF (ActPos > ArmPos[i]) THEN
				CheckRaised := INT_TO_USINT(i) ;
				EXIT ;
			END_IF
		END_FOR
	END_IF

	//RESET OUTPUTS
	FOR i := 0 TO 5 DO
		OUT[i]:= FALSE ;
	END_FOR

	//REQUIREMENTS FOR ARMS TO HOLD UP
	IF(Raise) OR(HiVol) THEN
		CASE CheckRaised OF
			0:	//NO ARMS UP
				UpDone := TRUE ;
			1:	//1 ARM UP
				OUT[1] := TRUE ;
			2:	//2 ARMS UP
				OUT[1] := TRUE ;
				OUT[2] := TRUE ;
			3:	//3 ARMS UP
				OUT[1] := TRUE ;
				OUT[2] := TRUE ;
				OUT[3] := TRUE ;
			4:	//4 ARMS UP
				OUT[1] := TRUE ;
				OUT[2] := TRUE ;
				OUT[3] := TRUE ;
				OUT[4] := TRUE ;
			5:	//5 ARMS UP
				OUT[1] := TRUE ;
				OUT[2] := TRUE ;
				OUT[3] := TRUE ;
				OUT[4] := TRUE ;
				OUT[5] := TRUE ;
		END_CASE
	END_IF

	//VERFIY SELECTED ARMS ARE IN THE UP POSITION
	IF(Raise) AND NOT(UpDone) THEN
		FOR i := 1 TO (CheckRaised * 2) DO
			IF NOT(Up[i]) THEN
				EXIT	;
			ELSIF (i = (CheckRaised * 2)) THEN
				UpDone := TRUE ;
			END_IF
		END_FOR
	END_IF

	//RESET CONDITIONS BEFORE NEXT SEEK AND FIND
	IF NOT(Raise) THEN
		CheckRaised := 0 ;
		UpDone :=	FALSE ;
	END_IF

END_FUNCTION_BLOCK
```

#### NozzleControl.st
```iecst
(********************************************************************
* COPYRIGHT ASHTON INDUSTRIAL SALES LTD. 2024
********************************************************************
* LIBRARY: Lib_Ashton
* FILE:  NozzleControl.st
* AUTHOR: NE
********************************************************************
* IMPLEMENTATION OF LIBRARY Lib_Ashton
 ********************************************************************)

//SPRAY NOZZLE CONTROL
FUNCTION_BLOCK NozzleControl

	// SPRAY NOZZLE START UP CONTROL STOP
	Nozzle.PurgeCount := NozzlePerm.PurgeCount;
	Nozzle.VacuumStopDelay := UDINT_TO_DINT(VacuumStopDelay/20);
	Nozzle.NozzleOpenDelay := NozzlePerm.OpenDelay/20;
	CASE Nozzle.Seq OF
		NC_Idle:
			Spray := FALSE;
			Nozzle.CountPurge := 0;
			IF(AutoStart)THEN
				Nozzle.Seq := NC_Open;
				Nozzle.Delay := 0;
			END_IF
		NC_Open:
			Spray := TRUE;
			Nozzle.Delay := Nozzle.Delay + 1;
			IF(Nozzle.Delay > 25)THEN
				Nozzle.Seq := NC_Close;
				Nozzle.Delay := 0;
			END_IF
		NC_Close:
			Spray := FALSE;
			Nozzle.Delay := Nozzle.Delay + 1;
			IF(Nozzle.Delay > 25)THEN
				Nozzle.CountPurge := Nozzle.CountPurge + 1;
				IF(Nozzle.CountPurge >= Nozzle.PurgeCount)THEN
					Nozzle.Seq := NC_CleanDone;
					IdleOpenTON.IN := FALSE;
					IdleIntervalTON.IN := TRUE;
				ELSE
					Nozzle.Seq := NC_Open;
					Nozzle.Delay := 0;
				END_IF
			END_IF
		NC_CleanDone:
			//LINE RUNNING SPRAY CONTROL
			Spray := FALSE;
			FOR TrackIndex := 0 TO 6 DO
				IF(Track[TrackIndex])THEN
					Spray := TRUE;
					SequenceIO := IO_IDLE;
					IdleIntervalTON.IN := FALSE;
					IdleOpenTON.IN := FALSE;
					EXIT;
				ELSE
					//DELAY FOR VALVE OPENING WHEN IDLE
					CASE SequenceIO OF
						IO_IDLE:
							SequenceIO := IO_INTERVAL;
							IdleIntervalTON.IN := FALSE;
							IdleOpenTON.IN := FALSE;
						IO_INTERVAL:
							Spray := FALSE;
							IdleIntervalTON.IN := TRUE;
							IdleOpenTON.IN := FALSE;
							IF(IdleIntervalTON.Q)THEN
								SequenceIO := IO_OPEN;
							END_IF
						IO_OPEN:
							Spray := TRUE;
							IdleIntervalTON.IN := FALSE;
							IdleOpenTON.IN := TRUE;
							IF(IdleOpenTON.Q)THEN
								SequenceIO := IO_INTERVAL;
							END_IF
					END_CASE
				END_IF
			END_FOR
			CASE PreTracking OF
				0:
				1:
					Spray := (PreTrack[1]) AND NOT(PreTrack[0]);
				2:
					Spray := (PreTrack[1] OR PreTrack[2]) AND NOT(PreTrack[0]);
			END_CASE
			//WAIT FOR CONTROL STOP
			IF NOT(Control)THEN
				Nozzle.Delay := 0;
				Nozzle.Seq := NC_ControlStop1;
			END_IF
			IF NOT(AutoStart)THEN
				Nozzle.Seq := NC_ControlStop2;
			END_IF
		NC_ControlStop1:
			Spray := TRUE;
			Nozzle.Delay := Nozzle.Delay + 1;
			IF(Nozzle.Delay > Nozzle.VacuumStopDelay)THEN
				Nozzle.Delay := 0;
				Nozzle.Seq := NC_ControlStop2;
			END_IF
		NC_ControlStop2:
			Spray := TRUE;
			Nozzle.Delay := Nozzle.Delay + 1;
			IF(Nozzle.Delay > Nozzle.NozzleOpenDelay)THEN
				Nozzle.Delay := 0;
				Nozzle.Seq := NC_Idle;
			END_IF
			ControlStop := ControlStop + 1;
	END_CASE
	IdleOpenTON.PT := t#10s;
	IdleOpenTON ();
	IdleIntervalTON.PT := t#2m30s;
	IdleIntervalTON ();
	IF(TransportMode)THEN
		Spray := FALSE;
	END_IF

END_FUNCTION_BLOCK
```

#### SeamersSMProIIFB.st
```iecst
(********************************************************************
* COPYRIGHT ASHTON INDUSTRIAL SALES LTD. OCT 2024
********************************************************************
* LIBRARY: Lib_Ashton
* FILE: SeamersSMProIIFB.st
* AUTHOR: NE
********************************************************************
* IMPLEMENTATION OF LIBRARY Lib_Ashton
 ********************************************************************)

//SEAMERS START UP AUTO SEQUENCE AND CONTROL SMPRO
FUNCTION_BLOCK SeamersSMProIIFB

	//ENABLE AUTO START SEQUENCE BUTTON ON SCREEN
	IF(Enable[1]) AND(Enable[2]) AND NOT(AutoStart[1]) AND NOT(AutoStart[2])THEN
		StartAllDisp := FB_SHOW;
	ELSE
		StartAllDisp := FB_HIDE;
	END_IF

	//=========================================================
	// sequenced start of seamer 1 process motors and pumps
	//=========================================================
	CASE AutoStart1 OF
		//=======================================================
		SS_Reset:
			Belt1TON.IN := FALSE;
			Belt2TON.IN := FALSE;
			Belt3TON.IN := FALSE;
			Belt4TON.IN := FALSE;
			Belt9TON.IN := FALSE;
			Belt10TON.IN := FALSE;
			Vac1TON.IN := FALSE;
			Vac2TON.IN := FALSE;
			Extract1TON.IN := FALSE;
			Extract2TON.IN := FALSE;
			BeltOUT[1] := FALSE;
			BeltOUT[2] := FALSE;
			BeltOUT[3] := FALSE;
			BeltOUT[4] := FALSE;
			BeltOUT[9] := FALSE;
			BeltOUT[10] := FALSE;
			VacOUT[1] := FALSE;
			VacOUT[2] := FALSE;
			ExtractionOUT[1] := FALSE;
			ExtractionOUT[2] := FALSE;
			Latch := FALSE;
			DoneOUT[1] := FALSE;

			IF NOT(Enable[1]) THEN
				DoneOUT[1] := TRUE;
			END_IF

			IF(AutoStart[0]) AND(LatchES) AND(AutoStart2 = SS_Started) THEN
				AutoStart[1] := TRUE;
			ELSIF(AutoStart[0]) AND(Control.Achieved) THEN
				AutoStart[1] := TRUE;
				Latch := TRUE;
			END_IF

			IF(TransportMode)THEN
				AutoStart1 := SS_VacuumPump1;
			ELSE
				AutoStart1 := SS_Ready;
			END_IF
		//=======================================================
		SS_Ready:
			IF(AutoStart[1])THEN
				AutoStart1 := SS_BeltMotor1;
			END_IF
		//=======================================================
		SS_BeltMotor1:
			BeltOUT[1] := TRUE;
			Belt1TON.IN := TRUE;
			IF (Belt1TON.Q)THEN
				AutoStart1 := SS_BeltMotor2;
			END_IF
		//=======================================================
		SS_BeltMotor2:
			BeltOUT[2] := TRUE;
			Belt2TON.IN := TRUE;
			IF(Belt2TON.Q)THEN
				AutoStart1 := SS_BeltMotor3;
			END_IF
		//=======================================================
		SS_BeltMotor3:
			BeltOUT[3] := TRUE;
			Belt3TON.IN := TRUE;
			IF (Belt3TON.Q)THEN
				AutoStart1 := SS_BeltMotor4;
			END_IF
		//=======================================================
		SS_BeltMotor4:
			BeltOUT[4] := TRUE;
			Belt4TON.IN := TRUE;
			IF(Intercept1 < ID_Open) AND((AutoStart2 = SS_Reset) OR(AutoStart2 = SS_BeltMotor4) OR(AutoStart2 = SS_Started))THEN
				IF(Belt4TON.Q)THEN
					AutoStart1 := SS_VacuumPump1;
				END_IF
			END_IF
		//=======================================================
		SS_VacuumPump1:
			VacOUT[1] := TRUE;
			Vac1TON.IN := TRUE;
			IF (Vac1TON.Q)THEN
				AutoStart1 := SS_VacuumPump2;
			END_IF
		//=======================================================
		SS_VacuumPump2:
			VacOUT[2] := TRUE;
			Vac2TON.IN := TRUE;
			IF(Vac2TON.Q)THEN
				IF(Shaker)THEN
					AutoStart1 := SS_Extraction1;
				ELSE
					AutoStart1 := SS_Started;
					IF(TransportMode)THEN
						AutoStart1 := SS_TransportMode;
						AutoStart2 := SS_VacuumPump1;
					ELSE
						AutoStart1 := SS_Started;
					END_IF
				END_IF
				IF(Latch)THEN
					AutoStart2 := SS_Reset;
					AutoStart[2] := TRUE;
				END_IF
			END_IF
		//=======================================================
		SS_Extraction1:
			ExtractionOUT[1] := TRUE;
			Extract1TON.IN := TRUE;
			IF(Extract1TON.Q)THEN
				AutoStart1 := SS_Extraction2;
			END_IF;
		//=======================================================
		SS_Extraction2:
			ExtractionOUT[2] := TRUE;
			Extract2TON.IN := TRUE;
			IF(Extract2TON.Q)THEN
				AutoStart1 := SS_Started;
			END_IF;
		//=======================================================
		SS_Started:
			DoneOUT[1] := TRUE;
			AutoStart[0] := FALSE;
			IF NOT((Enable[1]) OR (AutoStart[1]))THEN
				AutoStart1 := SS_Reset;
			END_IF

			IF(AutoStart2 > SS_Reset)THEN
				Latch := FALSE;
			END_IF

			//stop/start extraction when shaking
			ExtractionOUT[1] := NOT(Shaker);
			ExtractionOUT[2] := NOT(Shaker);
		//=======================================================
		SS_TransportMode:

	END_CASE

	Belt1TON.PT := PresetSys.Belt;
	Belt1TON ();
	Belt2TON.PT := PresetSys.Belt;
	Belt2TON ();
	Belt3TON.PT := PresetSys.Belt;
	Belt3TON ();
	Belt4TON.PT := PresetSys.Belt;
	Belt4TON ();
	Vac1TON.PT := PresetSys.Vac;
	Vac1TON ();
	Vac2TON.PT := PresetSys.Vac;
	Vac2TON ();
	Extract1TON.PT := PresetSys.Extraction;
	Extract1TON ();
	Extract2TON.PT := PresetSys.Extraction;
	Extract2TON ();

	// reset if motor starter trip detected
	IF(AutoStart[1])THEN
		FOR i:= 0 TO 9 DO
			IF(Trips[i])THEN
				AutoStart1 := SS_Reset;
				EXIT;
			END_IF
		END_FOR
	END_IF

	// reset sequence if buttons changed on terminal
	IF NOT(Enable[1]) OR NOT(Control.Achieved) OR(Detension)THEN
		AutoStart[1] := FALSE;
		AutoStart[0] := FALSE;
	END_IF

	IF NOT(AutoStart[1]) AND NOT(TransportMode)THEN
		AutoStart[1] := FALSE;
		AutoStart1 := SS_Reset;
	END_IF

	IF(TransportMode) AND NOT(Control.Achieved)THEN
		AutoStart[1] := FALSE;
		AutoStart1 := SS_Reset;
	END_IF

	//=========================================================
	// sequenced start of seamer 2 process motors and pumps
	//=========================================================
	CASE AutoStart2 OF
		//=======================================================
		SS_Reset:
			Belt5TON.IN := FALSE;
			Belt6TON.IN := FALSE;
			Belt7TON.IN := FALSE;
			Belt8TON.IN := FALSE;
			Belt11TON.IN := FALSE;
			Belt12TON.IN := FALSE;
			Vac3TON.IN := FALSE;
			Vac4TON.IN := FALSE;
			Extract3TON.IN := FALSE;
			Extract4TON.IN := FALSE;
			BeltOUT[5] := FALSE;
			BeltOUT[6] := FALSE;
			BeltOUT[7] := FALSE;
			BeltOUT[8] := FALSE;
			BeltOUT[11] := FALSE;
			BeltOUT[12] := FALSE;
			VacOUT[3] := FALSE;
			VacOUT[4] := FALSE;
			ExtractionOUT[3] := FALSE;
			ExtractionOUT[4] := FALSE;
			LatchES := FALSE;
			DoneOUT[2] := FALSE;

			IF NOT(Enable[2]) THEN
				DoneOUT[2] := TRUE;
			END_IF

			IF(AutoStart[0]) AND(Control.ESClear)THEN
				AutoStart[2] := TRUE;
				LatchES := TRUE;
			ELSIF(Latch) AND(AutoStart1 = SS_Started)THEN
				AutoStart[2] := TRUE;
			END_IF
			IF(TransportMode)THEN
				AutoStart2 := SS_VacuumPump1;
			ELSE
				AutoStart2 := SS_Ready;
			END_IF
		//=======================================================
		SS_Ready:
			IF(AutoStart[2])THEN
				AutoStart2 := SS_BeltMotor1;
			END_IF
		//=======================================================
		SS_BeltMotor1:
			BeltOUT[5] := TRUE;
			Belt5TON.IN := TRUE;
			IF (Belt5TON.Q)THEN
				AutoStart2 := SS_BeltMotor2;
			END_IF
		//=======================================================
		SS_BeltMotor2:
			BeltOUT[6] := TRUE;
			Belt6TON.IN := TRUE;
			IF(Belt6TON.Q)THEN
				AutoStart2 := SS_BeltMotor3;
			END_IF
		//=======================================================
		SS_BeltMotor3:
			BeltOUT[7] := TRUE;
			Belt7TON.IN := TRUE;
			IF (Belt7TON.Q)THEN
				AutoStart2 := SS_BeltMotor4;
			END_IF
		//=======================================================
		SS_BeltMotor4:
			BeltOUT[8] := TRUE;
			Belt8TON.IN := TRUE;
			IF(Intercept2 < ID_Open) AND((AutoStart1 = SS_Reset) OR(AutoStart1 = SS_BeltMotor4) OR(AutoStart1 = SS_Started))THEN
				IF(Belt8TON.Q)THEN
					AutoStart2 := SS_VacuumPump1;
				END_IF
			END_IF
		//=======================================================
		SS_VacuumPump1:
			VacOUT[3] := TRUE;
			Vac3TON.IN := TRUE;
			IF (Vac3TON.Q)THEN
				AutoStart2 := SS_VacuumPump2;
			END_IF
		//=======================================================
		SS_VacuumPump2:
			VacOUT[4] := TRUE;
			IF(Vac4TON.Q)THEN
				IF(Shaker)THEN
					AutoStart2 := SS_Extraction1;
				ELSE
					AutoStart2 := SS_Started;
					IF(TransportMode)THEN
						AutoStart2 := SS_TransportMode;
					ELSE
						AutoStart2 := SS_Started;
					END_IF
				END_IF
				IF(LatchES)THEN
					AutoStart1 := SS_Reset;
				END_IF
			END_IF
		//=======================================================
		SS_Extraction1:
			ExtractionOUT[3] := TRUE;
			Extract3TON.IN := TRUE;
			IF(Extract3TON.Q)THEN
				AutoStart2 := SS_Extraction2;
			END_IF;
		//=======================================================
		SS_Extraction2:
			ExtractionOUT[4] := TRUE;
			Extract4TON.IN := TRUE;
			IF(Extract4TON.Q)THEN
				AutoStart2 := SS_Started;
			END_IF;
		//=======================================================
		SS_Started:
			DoneOUT[2] := TRUE;
			AutoStart[0] := FALSE;
			IF NOT((Enable[1]) OR (AutoStart[1]) OR(Enable[2]) OR (AutoStart[2]))THEN
				AutoStart2 := SS_Reset;
			END_IF

			IF(AutoStart1 > SS_Reset)THEN
				LatchES := FALSE;
			END_IF

			//stop/start extraction when shaking
			ExtractionOUT[3] := NOT(Shaker);
			ExtractionOUT[4] := NOT(Shaker);
		//=======================================================
		SS_TransportMode:

	END_CASE

	Belt5TON.PT := PresetSys.Belt;
	Belt5TON ();
	Belt6TON.PT := PresetSys.Belt;
	Belt6TON ();
	Belt7TON.PT := PresetSys.Belt;
	Belt7TON ();
	Belt8TON.PT := PresetSys.Belt;
	Belt8TON ();
	Vac3TON.PT := PresetSys.Vac;
	Vac3TON ();
	Vac4TON.IN := TRUE;
	Vac4TON.PT := PresetSys.Vac;
	Vac4TON ();
	Extract3TON.PT := PresetSys.Extraction;
	Extract3TON ();
	Extract4TON.PT := PresetSys.Extraction;
	Extract4TON ();

	// reset if motor starter trip detected
	IF(AutoStart[2])THEN
		FOR i:= 10 TO 19 DO
			IF(Trips[i])THEN
				AutoStart2 := SS_Reset;
				EXIT;
			END_IF
		END_FOR
	END_IF

	// reset sequence if buttons changed on terminal
	IF NOT(Enable[2]) OR NOT(Control.Achieved) OR(Detension)THEN
		AutoStart[2] := FALSE;
		AutoStart[0] := FALSE;
	END_IF

	IF NOT(AutoStart[2]) AND NOT(TransportMode)THEN
		AutoStart[2] := FALSE;
		AutoStart2 := SS_Reset;
	END_IF

	IF(TransportMode) AND NOT(Control.Achieved)THEN
		AutoStart[2] := FALSE;
		AutoStart2 := SS_Reset;
	END_IF

	//==========================================
	// vacuum pumop run on control after control off
	//==========================================
	CASE VacuumRunOn OF
		//=======================================================
		VR_Idle:
			IF(Control.Achieved) THEN
				VacuumRunOn := VR_Done;
			END_IF
			VacStopTON.IN := FALSE;
		//=======================================================
		VR_Running:
			VacOUT[1] := TRUE;
			VacOUT[2] := TRUE;
			VacOUT[3] := TRUE;
			VacOUT[4] := TRUE;
			VacStopTON.IN := TRUE;
			VacStopTON.PT := PresetSys.VacsStop;
			IF(VacStopTON.Q)THEN
				VacuumRunOn := VR_Idle;
			END_IF
		//=======================================================
		VR_Done:
			VacStopTON.IN := FALSE;
			IF NOT(Control.Achieved) AND((Enable[1]) OR(Enable[2])) THEN
				VacuumRunOn := VR_Running;
			END_IF;

	END_CASE;

	VacStopTON ();

	//WATER CONTROL
	//START CONDITIONS FOR WATER PUMPS
	PumpOUT[1] := FALSE;
	PumpOUT[2] := FALSE;
	IF (AutoStart[1]) OR(AutoStart[2]) OR(PumpOUT[0])THEN
		IF(Control.Achieved) AND NOT(Pump1TON.Q)THEN
			PumpOUT[1] := TRUE;
		ELSE
			PumpOUT[1] := FALSE;
		END_IF
		IF (Control.Achieved) AND NOT(Pump2TON.Q)THEN
			PumpOUT[2] := TRUE;
		ELSE
			PumpOUT[2] := FALSE;
		END_IF
	END_IF

	//FLOAT SWITCH CONTROL OF WATER PUMP
	Pump1TON.IN := NOT(Float[1]);
	Pump1TON.PT := PresetSys.Water[1];
	Pump1TON ();

	Pump2TON.IN := NOT(Float[2]);
	Pump2TON.PT := PresetSys.Water[1];
	Pump2TON ();

	//SCAVENGE PUMP
	IF (AutoStart[1]) OR(AutoStart[2]) OR(PumpOUT[0]) THEN
		Pump3TON.IN := TRUE ;
	ELSE
		Pump3TON.IN := FALSE ;
	END_IF
	//DELAY BEFORE SCAVENGE PUMP STARTS
	Pump3TON.PT	:= PresetSys.Water[3] ;
	Pump3TON ();

	IF (Pump3TON.Q) AND NOT (Pump4TON.Q) THEN
		PumpOUT[0]	:= 	TRUE	;
	ELSE
		PumpOUT[0]	:= 	FALSE	;
	END_IF

	//DELAY BEFORE SCAVENGE PUMP STOP
	Pump4TON.PT	:= PresetSys.Water[4] ;
	Pump4TON ();

	IF NOT(AutoStart[1]) AND NOT(AutoStart[2]) THEN
		Pump4TON.IN := TRUE ;
	ELSE
		Pump4TON.IN := FALSE ;
	END_IF
	//SPRAY NOZZLE VALVE
	IF (AutoStart[1]) OR(AutoStart[2])THEN
		ValveOUT[1] := TRUE;
	ELSE
		ValveOUT[1] := FALSE;
	END_IF

	//SCAVENGE PUMP VALVE
	//DELAY BEFORE SCAVENGE PUMP STARTS
	Scavenge.Open.PT := PresetSys.Water[3];
	Scavenge.Open ();

	//VALVE OPEN
	ValveOUT[2] := Scavenge.Open.M;

	IF(Scavenge.Open.Q)THEN
		Scavenge.Open.IN := FALSE;
		Scavenge.Interval.IN := TRUE;
	END_IF

	//DELAY FOR INTERVAL BETWEEN VALVE OPENING
	IF EDGEPOS(Control.Achieved)THEN
		Scavenge.Open.IN := FALSE;
		Scavenge.Interval.IN := TRUE;
	END_IF
	IF NOT(Control.Achieved)THEN
		Scavenge.Open.IN := FALSE;
		Scavenge.Interval.IN := FALSE;
	END_IF
	IF(Scavenge.Open.PT = t#0ms)THEN
		Scavenge.Open.IN := FALSE;
		Scavenge.Interval.IN := FALSE;
		ValveOUT[2] := FALSE;
	END_IF

	Scavenge.Interval.PT := PresetSys.Water[4];
	Scavenge.Interval ();

	IF(Scavenge.Interval.Q)THEN
		Scavenge.Interval.IN := FALSE;
		Scavenge.Open.IN := TRUE;
	END_IF

	BackGround.AutoStart := AutoStart;
	BackGround.Enable := Enable;
	BackGround.ED := EDOn;

	//=========================================================
	// delay for intercept draining
	//=========================================================
	CASE Intercept1 OF
		//=======================================================
		ID_Idle:
			InterceptInterval1TON.IN := FALSE;
			InterceptOpen1TON.IN := FALSE;
			IF(AutoStart1 >= SS_Started)THEN
				Intercept1 := ID_Interval;
			END_IF
		//=======================================================
		ID_Interval:
			InterceptOpen1TON.IN := FALSE;
			InterceptInterval1TON.IN := TRUE;
			IF(InterceptInterval1TON.Q)THEN
				IF NOT(SeekBlock[1])THEN
					DoneOUT[1] := FALSE;
				END_IF
				IF NOT(SeekBlock[1])THEN
					AutoStart1 := SS_BeltMotor4;
					Vac1TON.IN := FALSE;
					Vac2TON.IN := FALSE;
					VacOUT[1] := FALSE;
					VacOUT[2] := FALSE;
					Intercept1 := ID_Open;
				END_IF
			END_IF
		//=======================================================
		ID_Open:
			InterceptInterval1TON.IN := FALSE;
			InterceptOpen1TON.IN := TRUE;
			IF(InterceptOpen1TON.Q)THEN
				Intercept1 := ID_Interval;
			END_IF
	END_CASE

	InterceptInterval1TON.PT := InterceptInterval;
	InterceptInterval1TON ();
	InterceptOpen1TON.PT := InterceptOpen;
	InterceptOpen1TON ();

	IF NOT(Control.Achieved) OR(AutoStart1 = SS_Reset)THEN
		Intercept1 := ID_Idle;
	END_IF

	//=========================================================
	// delay for intercept draining
	//=========================================================
	CASE Intercept2 OF
		//=======================================================
		ID_Idle:
			InterceptInterval2TON.IN := FALSE;
			InterceptOpen2TON.IN := FALSE;
			IF(AutoStart2 >= SS_Started)THEN
				Intercept2 := ID_Interval;
			END_IF
		//=======================================================
		ID_Interval:
			InterceptOpen2TON.IN := FALSE;
			InterceptInterval2TON.IN := TRUE;
			IF(InterceptInterval2TON.Q)THEN
				IF NOT(SeekBlock[2]) THEN
					DoneOUT[2] := FALSE;
				END_IF
				IF NOT(SeekBlock[2])THEN
					AutoStart2 := SS_BeltMotor4;
					Vac3TON.IN := FALSE;
					Vac4TON.IN := FALSE;
					VacOUT[3] := FALSE;
					VacOUT[4] := FALSE;
					Intercept2 := ID_Open;
				END_IF
			END_IF
		//=======================================================
		ID_Open:
			InterceptInterval2TON.IN := FALSE;
			InterceptOpen2TON.IN := TRUE;
			IF(InterceptOpen2TON.Q)THEN
				Intercept2 := ID_Interval;
			END_IF
	END_CASE

	InterceptInterval2TON.PT := InterceptInterval;
	InterceptInterval2TON ();
	InterceptOpen2TON.PT := InterceptOpen;
	InterceptOpen2TON ();

	IF NOT(Control.Achieved) OR(AutoStart2 = SS_Reset)THEN
		Intercept2 := ID_Idle;
	END_IF

END_FUNCTION_BLOCK
```

### Package Logical/System - Background system control

### System.var - Package variables
```iecst
(********************************************************************
 * COPYRIGHT --
 ********************************************************************
 * Package: System
 * File: System.var
 * Author: nicke
 * Created: February, 2012
 ********************************************************************
 * Variables of package System
 ********************************************************************)
VAR
	GrindFB1M : GrindTime;
	GrindFB2M : GrindTime;
	GrindFB1 : GrindTime;
	GrindFB2 : GrindTime;
	RunTime1 : RunTime;
END_VAR
```

### Program Logical/System/Control (IEC) - Control section of program

#### ControlCyclic.st - Cyclic code
```iecst
(********************************************************************
 * COPYRIGHT --
 ********************************************************************
 * Program: Control
 * File: ControlCyclic.st
 * Author: nicke
 ********************************************************************
 * Implementation of program Control
 ********************************************************************)

PROGRAM _CYCLIC

	Control.BuzzerPT := PresetSys.Buzzer ;
	Control.Paused := Pause.Active ;
	Control.Alarm := SysTemp.Alarm ;
	Control.Warning := SysTemp.Warning ;
	Control.StandbyPT := PresetSys.Standby ;
	Control.CountIN[0] := Tracking00.Busy ;
	Control.CountIN[1] := Tracking01.Busy ;
	Control.CountIN[2] := Tracking10.Busy ;
	Control.CountIN[3] := Tracking11.Busy ;
	Control.CountIN[4] := Tracking20.Busy ;
	Control.CountIN[5] := Tracking30.Busy ;
	Control.CountIN[6] := Tracking40.Busy ;
	Control.CountIN[7] := Tracking41.Busy ;
	Control.CountIN[8] := Tracking50.Busy ;
	Control.CountIN[9] := Tracking60.Busy ;
	Control.CountIN[10] := Tracking70.Busy ;
	Control.CountIN[11] := Tracking51.Busy ;

	Control ();

	Control.EStop2 := Control.EStop1 ;

END_PROGRAM
```

### Program Logical/System/Seamers (IEC) - Seaming motor control
